# B&R Automation Studio project CControl_Gschneitner (part 15)

#### Main.st - Init, cyclic, exit code
```iecst
PROGRAM _INIT

	hmiStatus.NameSteuerung	:= 6; //= LaTronic CControl 2.07

END_PROGRAM

PROGRAM _CYCLIC

	//Bei Konfiguration 4.07 -> Text auf Login-Seite anpassen, Option Entfeuchter ausschalten

	hmiParameter.Ausstattung.Entfeuchter := FALSE;
	hmiParameter.Ausstattung.Bypassklappe := FALSE;
	hmiParameter.Ausstattung.Box3 := FALSE;
	hmiParameter.Ausstattung.Box4 := FALSE;
	hmiParameter.Ausstattung.Box5 := FALSE;
	hmiParameter.Ausstattung.Box6 := FALSE;

	IF hmiParameter.Ausstattung.Abluftklappe THEN
		hmiParameter.Ausstattung.Abluftventilator := FALSE;
	ELSIF hmiParameter.Ausstattung.Abluftventilator THEN
		hmiParameter.Ausstattung.Abluftklappe := FALSE;
	END_IF

	//Zeitticks generieren
	fbLascoZdxx_0(IN 	:= Echtzeit.Sekunde);
	sekTick				:= fbLascoZdxx_0.Q;

	//=========================================================================================================================================================
	//IO-Zuweisung LaTronic CControl 4.07
	//=========================================================================================================================================================

	//Kein Testbetrieb
	IF (gAktModus <> IOTEST) THEN

		//MODUL 01 - BR7300 Busempfänger **********************************************************************************************************************
		brModul01;

		//MODUL 02 - CM8281 ***********************************************************************************************************************************
		//*****************************************************************************************************************************************************
		diVentilator1InBetrieb	:= cmModul02.di01;
		di24VDCinternIstOk		:= cmModul02.di02;
		//Reserve				:= cmModul02.di03;
		//Reserve				:= cmModul02.di04;

		cmModul02.do01			:= doVentilator1Ein;
		cmModul02.do02			:= doTrocknungInBetrieb;

		//Eingangssignale filtern
		IF sekTick THEN
			LCRMovAvgFlt_0(enable := TRUE, x := cmModul02.ai01, base := Betriebsparameter.Sensoren.FilterzeitFrischluft);
		END_IF

		//Frischluft Temperatur
		LCRLimScal_0(x := LCRMovAvgFlt_0.y, x1 := 0, y1 := Betriebsparameter.Sensoren.FrischlTempMessberMin,
		x2 := 32767, y2 := Betriebsparameter.Sensoren.FrischlTempMessberMax);
		aiFrischluftTemperatur		:= LCRLimScal_0.y + Betriebsparameter.Sensoren.OffsetFrischluftTemp;

		//Drehzahlvorgabe FU Ventilator 1
		LCRLimScal_0(x := aoDrehzahlvorgVentilator1, x1 := Betriebsparameter.Ventilator1.DrehzahlMin, y1 := 0,
		x2 := Betriebsparameter.Ventilator1.DrehzahlMax, y2 := 32767);
		cmModul02.ao01				:= REAL_TO_INT(LCRLimScal_0.y);

		//MODUL 03 - CM8281 ***********************************************************************************************************************************
		//*****************************************************************************************************************************************************
		diBox1Offen				:= cmModul03.di01;
		diBox1Geschl			:= cmModul03.di02;
		diBox2Offen				:= cmModul03.di03;
		diBox2Geschl			:= cmModul03.di04;

		cmModul03.do01			:= doFreigabeBox1;
		cmModul03.do02			:= doFreigabeBox2;

		//Eingangssignale filtern
		IF sekTick THEN
			LCRMovAvgFlt_1(enable := TRUE, x := cmModul03.ai01, base := Betriebsparameter.Sensoren.FilterzeitFrischluft);
		END_IF

		//Frischluft rel. Feuchte
		LCRLimScal_0(x := LCRMovAvgFlt_1.y, x1 := 0, y1 := Betriebsparameter.Sensoren.FrischlFeuchteMessberMin,
		x2 := 32767, y2 := Betriebsparameter.Sensoren.FrischlFeuchteMessberMax);
		aiFrischluftFeuchte		:= LCRLimScal_0.y + Betriebsparameter.Sensoren.OffsetFrischluftFeuchte;

		//Temperaturvorgabe Warmluftofen
		LCRLimScal_0(x := aoTemperaturvorgWarmluftofen, x1 := 0, y1 := 0,
		x2 := 100, y2 := 32767);
		cmModul03.ao01				:= REAL_TO_INT(LCRLimScal_0.y);

		//MODUL 04 - CM8281 ***********************************************************************************************************************************
		//*****************************************************************************************************************************************************
		diVentilator2InBetrieb			:= cmModul04.di01;
		diDrehzahlbegrVentilator1		:= cmModul04.di02;
		diDrehzahlbegrVentilator2		:= cmModul04.di03;
		//Reserve						:= cmModul04.di04;

		cmModul04.do01					:= doTrocknungStoerung;
		cmModul04.do02					:= doVentilator2Ein;

		//Eingangssignale filtern
		IF sekTick THEN
			LCRMovAvgFlt_2(enable := TRUE, x := cmModul04.ai01, base := Betriebsparameter.Sensoren.FilterzeitTrockenluft);
		END_IF

		//Trockenluft Temperatur
		LCRLimScal_0(x := LCRMovAvgFlt_2.y, x1 := 0, y1 := Betriebsparameter.Sensoren.TrockenlTempMessberMin,
		x2 := 32767, y2 := Betriebsparameter.Sensoren.TrockenlTempMessberMax);
		aiTrockenluftTemperatur		:= LCRLimScal_0.y + Betriebsparameter.Sensoren.OffsetTrockenluftTemp;

		//Drehzahlvorgabe FU Ventilator 2
		LCRLimScal_0(x := aoDrehzahlvorgVentilator2, x1 := Betriebsparameter.Ventilator2.DrehzahlMin, y1 := 0,
		x2 := Betriebsparameter.Ventilator2.DrehzahlMax, y2 := 32767);
		cmModul04.ao01				:= REAL_TO_INT(LCRLimScal_0.y);

		//MODUL 05 - CM8281 ***********************************************************************************************************************************
		//*****************************************************************************************************************************************************
		diWarmluftofenInBetrieb		:= cmModul05.di01;
		diScheitholzofenInBetrieb	:= cmModul05.di02;
		//Reserve					:= cmModul05.di03;
		//Reserve					:= cmModul05.di04;

		cmModul05.do01				:= doWarmluftofenEin;
		cmModul05.do02				:= doHeizregisterEin;

		//Eingangssignale filtern
		IF sekTick THEN
			LCRMovAvgFlt_3(enable := TRUE, x := cmModul05.ai01, base := Betriebsparameter.Sensoren.FilterzeitTrockenluft);
		END_IF

		//Trockenluft rel. Feuchte
		LCRLimScal_0(x := LCRMovAvgFlt_3.y, x1 := 0, y1 := Betriebsparameter.Sensoren.TrockenlFeuchteMessberMin,
		x2 := 32767, y2 := Betriebsparameter.Sensoren.TrockenlFeuchteMessberMax);
		aiTrockenluftFeuchte		:= LCRLimScal_0.y + Betriebsparameter.Sensoren.OffsetTrockenluftFeuchte;

		//Leistungsvorgabe Heizregister
		LCRLimScal_0(x := aoLeistungsvorgHeizregister, x1 := 0.0, y1 := 0, x2 := 100.0, y2 := 32767);
		cmModul05.ao01				:= REAL_TO_INT(LCRLimScal_0.y);

		//MODUL 06 - CM8281 ***********************************************************************************************************************************
		//*****************************************************************************************************************************************************
		diBox3Offen				:= cmModul06.di01;
		diBox3Geschl			:= cmModul06.di02;
		diBox4Offen				:= cmModul06.di03;
		diBox4Geschl			:= cmModul06.di04;

		cmModul06.do01			:= doFreigabeBox3;
		cmModul06.do02			:= doFreigabeBox4;

		//Eingangssignale filtern
		IF sekTick THEN
			LCRMovAvgFlt_4(enable := TRUE, x := cmModul06.ai01, base := Betriebsparameter.Sensoren.FilterzeitAbluft);
		END_IF

		//Abluft Temperatur
		LCRLimScal_0(x := LCRMovAvgFlt_4.y, x1 := 0, y1 := Betriebsparameter.Sensoren.AbluftTempMessberMin,
		x2 := 32767, y2 := Betriebsparameter.Sensoren.AbluftTempMessberMax);
		aiAbluftTemperatur		:= LCRLimScal_0.y + Betriebsparameter.Sensoren.OffsetAbluftTemp;

		//Analogausgang
		cmModul06.ao01				:= 0;	//Reserve

		//MODUL 07 - CM8281 ***********************************************************************************************************************************
		//*****************************************************************************************************************************************************
		diBox5Offen				:= cmModul07.di01;
		diBox5Geschl			:= cmModul07.di02;
		diBox6Offen				:= cmModul07.di03;
		diBox6Geschl			:= cmModul07.di04;

		cmModul07.do01			:= doFreigabeBox5;
		cmModul07.do02			:= doFreigabeBox6;

		//Eingangssignale filtern
		IF sekTick THEN
			LCRMovAvgFlt_5(enable := TRUE, x := cmModul07.ai01, base := Betriebsparameter.Sensoren.FilterzeitAbluft);
		END_IF

		//Abluft rel. Feuchte
		LCRLimScal_0(x := LCRMovAvgFlt_5.y, x1 := 0, y1 := Betriebsparameter.Sensoren.AbluftFeuchteMessberMin,
		x2 := 32767, y2 := Betriebsparameter.Sensoren.AbluftFeuchteMessberMax);
		aiAbluftFeuchte		:= LCRLimScal_0.y + Betriebsparameter.Sensoren.OffsetAbluftFeuchte;

		//Analogausgang
		cmModul07.ao01				:= 0;	//Reserve

		//MODUL 08 - CM8281 ***********************************************************************************************************************************
		//*****************************************************************************************************************************************************
		diAbluftventInBetrieb	:= cmModul08.di01;
		//Reserve				:= cmModul08.di02;
		//Reserve				:= cmModul08.di03;
		//Reserve				:= cmModul08.di04;

		cmModul08.do01			:= doBrandschutzklappeAuf;
		cmModul08.do02			:= doAbluftventilatorEin;

		//Eingangssignale filtern
		IF sekTick THEN
			LCRMovAvgFlt_6(enable := TRUE, x := cmModul08.ai01, base := Betriebsparameter.Sensoren.FilterzeitDachluft);
		END_IF

		//Dachluft Temperatur
		LCRLimScal_0(x := LCRMovAvgFlt_6.y, x1 := 0, y1 := Betriebsparameter.Sensoren.DachTempMessberMin,
		x2 := 32767, y2 := Betriebsparameter.Sensoren.DachTempMessberMax);
		aiDachluftTemperatur		:= LCRLimScal_0.y + Betriebsparameter.Sensoren.OffsetDachTemp;

		//Drehzahlvorgabe Abluftventilator
		LCRLimScal_0(x := aoDrehzahlvorgAbluftventilator, x1 := Betriebsparameter.Abluftventilator.DrehzahlMin, y1 := 0,
		x2 := Betriebsparameter.Abluftventilator.DrehzahlMax, y2 := 32767);
		cmModul08.ao01				:= REAL_TO_INT(LCRLimScal_0.y);

		//MODUL 09 - CM8281 ***********************************************************************************************************************************
		//*****************************************************************************************************************************************************
		diAbluftklappeOffen		:= cmModul09.di01;
		diAbluftklappeGeschl	:= cmModul09.di02;
		//Reserve				:= cmModul09.di03;
		//Reserve				:= cmModul09.di04;

		cmModul09.do01			:= doAbluftklappeFreigabe;
		cmModul09.do02			:= FALSE;	//Reserve

		//Eingangssignale filtern
		IF sekTick THEN
			LCRMovAvgFlt_7(enable := TRUE, x := cmModul09.ai01, base := Betriebsparameter.Sensoren.FilterzeitDachluft);
		END_IF

		//Dachluft rel. Feuchte
		LCRLimScal_0(x := LCRMovAvgFlt_7.y, x1 := 0, y1 := Betriebsparameter.Sensoren.DachFeuchteMessberMin,
		x2 := 32767, y2 := Betriebsparameter.Sensoren.DachFeuchteMessberMax);
		aiDachluftFeuchte		:= LCRLimScal_0.y + Betriebsparameter.Sensoren.OffsetDachFeuchte;

		//Analogausgang
		cmModul09.ao01				:= 0;	//Reserve

		//MODUL 10 - CM8281 ***********************************************************************************************************************************
		//*****************************************************************************************************************************************************
		diUmschaltklappe1Offen		:= cmModul10.di01;
		diUmschaltklappe1Geschl		:= cmModul10.di02;
		diUmschaltklappe2Offen		:= cmModul10.di03;
		diUmschaltklappe2Geschl		:= cmModul10.di04;

		cmModul10.do01				:= doUmluftklappe1Freigabe;
		cmModul10.do02				:= doUmluftklappe2Freigabe;

		//Eingangssignale filtern
		IF sekTick THEN
			LCRMovAvgFlt_8(enable := TRUE, x := cmModul10.ai01, base := Betriebsparameter.Sensoren.FilterzeitLuftgeschwindigkeit);
		END_IF

		//Luftgeschwindigkeit
		LCRLimScal_0(x := LCRMovAvgFlt_8.y, x1 := 0, y1 := Betriebsparameter.Sensoren.LuftgeschwMessberMin,
		x2 := 32767, y2 := Betriebsparameter.Sensoren.LuftgeschwMessberMax);
		aiLuftgeschwindigkeit		:= LCRLimScal_0.y + Betriebsparameter.Sensoren.OffsetLuftgeschw;

		//Analogausgang
		cmModul10.ao01				:= 0;	//Reserve

		//MODUL 11 - CM8281 ***********************************************************************************************************************************
		//*****************************************************************************************************************************************************
		diNotstromaggregatInBetrieb		:= cmModul11.di01;
		//Reserve						:= cmModul11.di02;
		//Reserve						:= cmModul11.di03;
		//Reserve						:= cmModul11.di04;

		cmModul11.do01					:= doNotstromaggregatEin;
		cmModul11.do02					:= FALSE;	//Reserve

		//Eingangssignale filtern
		IF sekTick THEN
			LCRMovAvgFlt_9(enable := TRUE, x := cmModul11.ai01, base := Betriebsparameter.Sensoren.FilterzeitKanaldruck);
		END_IF

		//Differenzdruck
		LCRLimScal_0(x := LCRMovAvgFlt_9.y, x1 := 0, y1 := Betriebsparameter.Sensoren.KanaldruckMessberMin,
		x2 := 32767, y2 := Betriebsparameter.Sensoren.KanaldruckMessberMax);
		aiDifferenzdruck		:= LCRLimScal_0.y + Betriebsparameter.Sensoren.OffsetKanaldruck;

		//Analogausgang
		cmModul11.ao01				:= 0;	//Reserve

		//Modulstatus - Auswertung **********************************************************************************************************************************
		//***********************************************************************************************************************************************************

		//Modul 02 Frischluft Temperatur ****************************************************************************
		IF (cmModul02.StatusInput01.1 = FALSE AND cmModul02.StatusInput01.0 = TRUE) THEN
			diStatusFrischluftTempMin	:= TRUE;
		ELSE
			diStatusFrischluftTempMin	:= FALSE;
		END_IF
		IF (cmModul02.StatusInput01.1 = TRUE AND cmModul02.StatusInput01.0 = FALSE ) THEN
			diStatusFrischluftTempMax	 := TRUE;
		ELSE
			diStatusFrischluftTempMax	 := FALSE;
		END_IF

		//Modul 03 Frischluft rel. Feuchte ****************************************************************************
		IF (cmModul03.StatusInput01.1 = FALSE AND cmModul03.StatusInput01.0 = TRUE) THEN
			diStatusFrischluftFeuchteMin	:= TRUE;
		ELSE
			diStatusFrischluftFeuchteMin	:= FALSE;
		END_IF
		IF (cmModul03.StatusInput01.1 = TRUE AND cmModul03.StatusInput01.0 = FALSE ) THEN
			diStatusFrischluftFeuchteMax	 := TRUE;
		ELSE
			diStatusFrischluftFeuchteMax	 := FALSE;
		END_IF

		//Modul 04 Trockenluft Temperatur ****************************************************************************
		IF (cmModul04.StatusInput01.1 = FALSE AND cmModul04.StatusInput01.0 = TRUE) THEN
			diStatusTrockenluftTempMin	:= TRUE;
		ELSE
			diStatusTrockenluftTempMin	:= FALSE;
		END_IF
		IF (cmModul04.StatusInput01.1 = TRUE AND cmModul04.StatusInput01.0 = FALSE ) THEN
			diStatusTrockenluftTempMax	 := TRUE;
		ELSE
			diStatusTrockenluftTempMax	 := FALSE;
		END_IF

		//Modul 05 Trockenluft rel. Feuchte ****************************************************************************
		IF (cmModul05.StatusInput01.1 = FALSE AND cmModul05.StatusInput01.0 = TRUE) THEN
			diStatusTrockenluftFeuchteMin	:= TRUE;
		ELSE
			diStatusTrockenluftFeuchteMin	:= FALSE;
		END_IF
		IF (cmModul05.StatusInput01.1 = TRUE AND cmModul05.StatusInput01.0 = FALSE ) THEN
			diStatusTrockenluftFeuchteMax	 := TRUE;
		ELSE
			diStatusTrockenluftFeuchteMax	 := FALSE;
		END_IF

		//Modul 06 Abluft Temperatur ****************************************************************************
		IF (cmModul06.StatusInput01.1 = FALSE AND cmModul06.StatusInput01.0 = TRUE) THEN
			diStatusAbluftTempMin	:= TRUE;
		ELSE
			diStatusAbluftTempMin	:= FALSE;
		END_IF
		IF (cmModul06.StatusInput01.1 = TRUE AND cmModul06.StatusInput01.0 = FALSE ) THEN
			diStatusAbluftTempMax	 := TRUE;
		ELSE
			diStatusAbluftTempMax	 := FALSE;
		END_IF

		//Modul 07 Abluft rel. Feuchte ****************************************************************************
		IF (cmModul07.StatusInput01.1 = FALSE AND cmModul07.StatusInput01.0 = TRUE) THEN
			diStatusAbluftFeuchteMin	:= TRUE;
		ELSE
			diStatusAbluftFeuchteMin	:= FALSE;
		END_IF
		IF (cmModul07.StatusInput01.1 = TRUE AND cmModul07.StatusInput01.0 = FALSE ) THEN
			diStatusAbluftFeuchteMax	 := TRUE;
		ELSE
			diStatusAbluftFeuchteMax	 := FALSE;
		END_IF

		//Modul 08 Dachluft Temperatur ****************************************************************************
		IF (cmModul08.StatusInput01.1 = FALSE AND cmModul08.StatusInput01.0 = TRUE) THEN
			diStatusDachluftTempMin	:= TRUE;
		ELSE
			diStatusDachluftTempMin	:= FALSE;
		END_IF
		IF (cmModul08.StatusInput01.1 = TRUE AND cmModul08.StatusInput01.0 = FALSE ) THEN
			diStatusDachluftTempMax	 := TRUE;
		ELSE
			diStatusDachluftTempMax	 := FALSE;
		END_IF

		//Modul 09 Dachluft rel. Feuchte ****************************************************************************
		IF (cmModul09.StatusInput01.1 = FALSE AND cmModul09.StatusInput01.0 = TRUE) THEN
			diStatusDachluftFeuchteMin	:= TRUE;
		ELSE
			diStatusDachluftFeuchteMin	:= FALSE;
		END_IF
		IF (cmModul09.StatusInput01.1 = TRUE AND cmModul09.StatusInput01.0 = FALSE ) THEN
			diStatusDachluftFeuchteMax	 := TRUE;
		ELSE
			diStatusDachluftFeuchteMax	 := FALSE;
		END_IF

		//Modul 10 Luftgeschwindigkeit ****************************************************************************
		IF (cmModul10.StatusInput01.1 = FALSE AND cmModul10.StatusInput01.0 = TRUE) THEN
			diStatusLuftgeschwMin	:= TRUE;
		ELSE
			diStatusLuftgeschwMin	:= FALSE;
		END_IF
		IF (cmModul10.StatusInput01.1 = TRUE AND cmModul10.StatusInput01.0 = FALSE ) THEN
			diStatusLuftgeschwMax	:= TRUE;
		ELSE
			diStatusLuftgeschwMax	 := FALSE;
		END_IF
		IF ((cmModul10.StatusInput01.1 = TRUE AND cmModul10.StatusInput01.0 = TRUE) OR cmModul10.ai01 >= 32767) THEN
			diStatusLuftgeschwDrahtbruch := TRUE;
		ELSE
			diStatusLuftgeschwDrahtbruch := FALSE;
		END_IF

		//Modul 11 Differenzdruck ****************************************************************************
		IF (cmModul11.StatusInput01.1 = FALSE AND cmModul11.StatusInput01.0 = TRUE) THEN
			diStatusDifferenzdruckMin	:= TRUE;
		ELSE
			diStatusDifferenzdruckMin	:= FALSE;
		END_IF
		IF (cmModul11.StatusInput01.1 = TRUE AND cmModul11.StatusInput01.0 = FALSE ) THEN
			diStatusDifferenzdruckMax	 := TRUE;
		ELSE
			diStatusDifferenzdruckMax	 := FALSE;
		END_IF

		//Ausgänge Testbetrieb rücksetzen, wenn IO-Test nicht aktiv
		hmiIoTest.DigitalOut.doAbluftklappeFreigabe		:= FALSE;
		hmiIoTest.DigitalOut.doAbluftventilatorEin		:= FALSE;
		hmiIoTest.DigitalOut.doBrandschutzklappeAuf		:= FALSE;
		hmiIoTest.DigitalOut.doBypassklappeOeffnen		:= FALSE;
		hmiIoTest.DigitalOut.doFreigabeBox1				:= FALSE;
		hmiIoTest.DigitalOut.doFreigabeBox2				:= FALSE;
		hmiIoTest.DigitalOut.doFreigabeBox3				:= FALSE;
		hmiIoTest.DigitalOut.doFreigabeBox4				:= FALSE;
		hmiIoTest.DigitalOut.doFreigabeBox5				:= FALSE;
		hmiIoTest.DigitalOut.doFreigabeBox6				:= FALSE;
		hmiIoTest.DigitalOut.doHeizregisterEin			:= FALSE;
		hmiIoTest.DigitalOut.doKompressorEinModul1		:= FALSE;
		hmiIoTest.DigitalOut.doKompressorEinModul2		:= FALSE;
		hmiIoTest.DigitalOut.doMagnetventilEinModul1	:= FALSE;
		hmiIoTest.DigitalOut.doMagnetventilEinModul2	:= FALSE;
		hmiIoTest.DigitalOut.doNotstromaggregatEin		:= FALSE;
		hmiIoTest.DigitalOut.doOelsumpfheizungEinModul1	:= FALSE;
		hmiIoTest.DigitalOut.doOelsumpfheizungEinModul2	:= FALSE;
		hmiIoTest.DigitalOut.doTrocknungInBetrieb		:= FALSE;
		hmiIoTest.DigitalOut.doTrocknungStoerung		:= FALSE;
		hmiIoTest.DigitalOut.doUmluftklappe1Freigabe	:= FALSE;
		hmiIoTest.DigitalOut.doUmluftklappe2Freigabe	:= FALSE;
		hmiIoTest.DigitalOut.doVentilator1Ein			:= FALSE;
		hmiIoTest.DigitalOut.doVentilator2Ein			:= FALSE;
		hmiIoTest.DigitalOut.doWarmluftofenEin			:= FALSE;

		hmiIoTest.AnalogOut.aoDrehzahlvorgAbluftventilator	:= 0.0;
		hmiIoTest.AnalogOut.aoDrehzahlvorgKompressorModul1	:= 0.0;
		hmiIoTest.AnalogOut.aoDrehzahlvorgKompressorModul2	:= 0.0;
		hmiIoTest.AnalogOut.aoDrehzahlvorgVentilator1		:= 0.0;
		hmiIoTest.AnalogOut.aoDrehzahlvorgVentilator2		:= 0.0;
		hmiIoTest.AnalogOut.aoLeistungsvorgHeizregister		:= 0.0;
		hmiIoTest.AnalogOut.aoTemperaturvorgWarmluftofen	:= 0.0;

	//==============================================================================================================================================================================================================
	//Testbetrieb
	//==============================================================================================================================================================================================================
	ELSE

		//MODUL 01 - BR7300 Busempfänger **********************************************************************************************************************

		//MODUL 02 - CM8281 ***********************************************************************************************************************************
		//*****************************************************************************************************************************************************
		hmiIoTest.DigitalIn.diVentilator1InBetrieb	:= cmModul02.di01;
		hmiIoTest.DigitalIn.di24VDCinternIstOk		:= cmModul02.di02;
		//Reserve									:= cmModul02.di03;
		//Reserve									:= cmModul02.di04;

		cmModul02.do01			:= hmiIoTest.DigitalOut.doVentilator1Ein;
		cmModul02.do02			:= hmiIoTest.DigitalOut.doTrocknungInBetrieb;

		//Eingangssignale filtern
		IF sekTick THEN
			LCRMovAvgFlt_0(enable := TRUE, x := cmModul02.ai01, base := Betriebsparameter.Sensoren.FilterzeitFrischluft);
		END_IF

		//Frischluft Temperatur
		LCRLimScal_0(x := LCRMovAvgFlt_0.y, x1 := 0, y1 := Betriebsparameter.Sensoren.FrischlTempMessberMin,
		x2 := 32767, y2 := Betriebsparameter.Sensoren.FrischlTempMessberMax);
		hmiIoTest.AnalogIn.aiFrischluftTemperatur		:= LCRLimScal_0.y + Betriebsparameter.Sensoren.OffsetFrischluftTemp;

		//Drehzahlvorgabe FU Ventilator 1
		LCRLimScal_0(x := hmiIoTest.AnalogOut.aoDrehzahlvorgVentilator1, x1 := Betriebsparameter.Ventilator1.DrehzahlMin, y1 := 0,
		x2 := Betriebsparameter.Ventilator1.DrehzahlMax, y2 := 32767);
		cmModul02.ao01				:= REAL_TO_INT(LCRLimScal_0.y);

		//MODUL 03 - CM8281 ***********************************************************************************************************************************
		//*****************************************************************************************************************************************************
		hmiIoTest.DigitalIn.diBox1Offen				:= cmModul03.di01;
		hmiIoTest.DigitalIn.diBox1Geschl			:= cmModul03.di02;
		hmiIoTest.DigitalIn.diBox2Offen				:= cmModul03.di03;
		hmiIoTest.DigitalIn.diBox2Geschl			:= cmModul03.di04;

		cmModul03.do01			:= hmiIoTest.DigitalOut.doFreigabeBox1;
		cmModul03.do02			:= hmiIoTest.DigitalOut.doFreigabeBox2;

		//Eingangssignale filtern
		IF sekTick THEN
			LCRMovAvgFlt_1(enable := TRUE, x := cmModul03.ai01, base := Betriebsparameter.Sensoren.FilterzeitFrischluft);
		END_IF

		//Frischluft rel. Feuchte
		LCRLimScal_0(x := LCRMovAvgFlt_1.y, x1 := 0, y1 := Betriebsparameter.Sensoren.FrischlFeuchteMessberMin,
		x2 := 32767, y2 := Betriebsparameter.Sensoren.FrischlFeuchteMessberMax);
		hmiIoTest.AnalogIn.aiFrischluftFeuchte		:= LCRLimScal_0.y + Betriebsparameter.Sensoren.OffsetFrischluftFeuchte;

		//Temperaturvorgabe Warmluftofen
		LCRLimScal_0(x := hmiIoTest.AnalogOut.aoTemperaturvorgWarmluftofen, x1 := 0, y1 := 0,
		x2 := 100, y2 := 32767);
		cmModul03.ao01				:= REAL_TO_INT(LCRLimScal_0.y);

		//MODUL 04 - CM8281 ***********************************************************************************************************************************
		//*****************************************************************************************************************************************************
		hmiIoTest.DigitalIn.diVentilator2InBetrieb			:= cmModul04.di01;
		hmiIoTest.DigitalIn.diDrehzahlbegrVentilator1		:= cmModul04.di02;
		hmiIoTest.DigitalIn.diDrehzahlbegrVentilator2		:= cmModul04.di03;
		//Reserve											:= cmModul04.di04;

		cmModul04.do01					:= hmiIoTest.DigitalOut.doTrocknungStoerung;
		cmModul04.do02					:= hmiIoTest.DigitalOut.doVentilator2Ein;

		//Eingangssignale filtern
		IF sekTick THEN
			LCRMovAvgFlt_2(enable := TRUE, x := cmModul04.ai01, base := Betriebsparameter.Sensoren.FilterzeitTrockenluft);
		END_IF

		//Trockenluft Temperatur
		LCRLimScal_0(x := LCRMovAvgFlt_2.y, x1 := 0, y1 := Betriebsparameter.Sensoren.TrockenlTempMessberMin,
		x2 := 32767, y2 := Betriebsparameter.Sensoren.TrockenlTempMessberMax);
		hmiIoTest.AnalogIn.aiTrockenluftTemperatur		:= LCRLimScal_0.y + Betriebsparameter.Sensoren.OffsetTrockenluftTemp;

		//Drehzahlvorgabe FU Ventilator 2
		LCRLimScal_0(x := hmiIoTest.AnalogOut.aoDrehzahlvorgVentilator2, x1 := Betriebsparameter.Ventilator2.DrehzahlMin, y1 := 0,
		x2 := Betriebsparameter.Ventilator2.DrehzahlMax, y2 := 32767);
		cmModul04.ao01				:= REAL_TO_INT(LCRLimScal_0.y);

		//MODUL 05 - CM8281 ***********************************************************************************************************************************
		//*****************************************************************************************************************************************************
		hmiIoTest.DigitalIn.diWarmluftofenInBetrieb		:= cmModul05.di01;
		hmiIoTest.DigitalIn.diScheitholzofenInBetrieb	:= cmModul05.di02;
		//Reserve										:= cmModul05.di03;
		//Reserve										:= cmModul05.di04;

		cmModul05.do01				:= hmiIoTest.DigitalOut.doWarmluftofenEin;
		cmModul05.do02				:= hmiIoTest.DigitalOut.doHeizregisterEin;

		//Eingangssignale filtern
		IF sekTick THEN
			LCRMovAvgFlt_3(enable := TRUE, x := cmModul05.ai01, base := Betriebsparameter.Sensoren.FilterzeitTrockenluft);
		END_IF

		//Trockenluft rel. Feuchte
		LCRLimScal_0(x := LCRMovAvgFlt_3.y, x1 := 0, y1 := Betriebsparameter.Sensoren.TrockenlFeuchteMessberMin,
		x2 := 32767, y2 := Betriebsparameter.Sensoren.TrockenlFeuchteMessberMax);
		hmiIoTest.AnalogIn.aiTrockenluftFeuchte		:= LCRLimScal_0.y + Betriebsparameter.Sensoren.OffsetTrockenluftFeuchte;

		//Leistungsvorgabe Heizregister
		LCRLimScal_0(x := hmiIoTest.AnalogOut.aoLeistungsvorgHeizregister, x1 := 0.0, y1 := 0, x2 := 100.0, y2 := 32767);
		cmModul05.ao01				:= REAL_TO_INT(LCRLimScal_0.y);

		//MODUL 06 - CM8281 ***********************************************************************************************************************************
		//*****************************************************************************************************************************************************
		hmiIoTest.DigitalIn.diBox3Offen				:= cmModul06.di01;
		hmiIoTest.DigitalIn.diBox3Geschl			:= cmModul06.di02;
		hmiIoTest.DigitalIn.diBox4Offen				:= cmModul06.di03;
		hmiIoTest.DigitalIn.diBox4Geschl			:= cmModul06.di04;

		cmModul06.do01			:= hmiIoTest.DigitalOut.doFreigabeBox3;
		cmModul06.do02			:= hmiIoTest.DigitalOut.doFreigabeBox4;

		//Eingangssignale filtern
		IF sekTick THEN
			LCRMovAvgFlt_4(enable := TRUE, x := cmModul06.ai01, base := Betriebsparameter.Sensoren.FilterzeitAbluft);
		END_IF

		//Abluft Temperatur
		LCRLimScal_0(x := LCRMovAvgFlt_4.y, x1 := 0, y1 := Betriebsparameter.Sensoren.AbluftTempMessberMin,
		x2 := 32767, y2 := Betriebsparameter.Sensoren.AbluftTempMessberMax);
		hmiIoTest.AnalogIn.aiAbluftTemperatur		:= LCRLimScal_0.y + Betriebsparameter.Sensoren.OffsetAbluftTemp;

		//Analogausgang
		cmModul06.ao01				:= 0;	//Reserve

		//MODUL 07 - CM8281 ***********************************************************************************************************************************
		//*****************************************************************************************************************************************************
		hmiIoTest.DigitalIn.diBox5Offen				:= cmModul07.di01;
		hmiIoTest.DigitalIn.diBox5Geschl			:= cmModul07.di02;
		hmiIoTest.DigitalIn.diBox6Offen				:= cmModul07.di03;
		hmiIoTest.DigitalIn.diBox6Geschl			:= cmModul07.di04;

		cmModul07.do01			:= hmiIoTest.DigitalOut.doFreigabeBox5;
		cmModul07.do02			:= hmiIoTest.DigitalOut.doFreigabeBox6;

		//Eingangssignale filtern
		IF sekTick THEN
			LCRMovAvgFlt_5(enable := TRUE, x := cmModul07.ai01, base := Betriebsparameter.Sensoren.FilterzeitAbluft);
		END_IF

		//Abluft rel. Feuchte
		LCRLimScal_0(x := LCRMovAvgFlt_5.y, x1 := 0, y1 := Betriebsparameter.Sensoren.AbluftFeuchteMessberMin,
		x2 := 32767, y2 := Betriebsparameter.Sensoren.AbluftFeuchteMessberMax);
		hmiIoTest.AnalogIn.aiAbluftFeuchte		:= LCRLimScal_0.y + Betriebsparameter.Sensoren.OffsetAbluftFeuchte;

		//Analogausgang
		cmModul07.ao01				:= 0;	//Reserve

		//MODUL 08 - CM8281 ***********************************************************************************************************************************
		//*****************************************************************************************************************************************************
		hmiIoTest.DigitalIn.diAbluftventInBetrieb	:= cmModul08.di01;
		//Reserve									:= cmModul08.di02;
		//Reserve									:= cmModul08.di03;
		//Reserve									:= cmModul08.di04;

		cmModul08.do01			:= hmiIoTest.DigitalOut.doBrandschutzklappeAuf;
		cmModul08.do02			:= hmiIoTest.DigitalOut.doAbluftventilatorEin;

		//Eingangssignale filtern
		IF sekTick THEN
			LCRMovAvgFlt_6(enable := TRUE, x := cmModul08.ai01, base := Betriebsparameter.Sensoren.FilterzeitDachluft);
		END_IF

		//Dachluft Temperatur
		LCRLimScal_0(x := LCRMovAvgFlt_6.y, x1 := 0, y1 := Betriebsparameter.Sensoren.DachTempMessberMin,
		x2 := 32767, y2 := Betriebsparameter.Sensoren.DachTempMessberMax);
		hmiIoTest.AnalogIn.aiDachluftTemperatur		:= LCRLimScal_0.y + Betriebsparameter.Sensoren.OffsetDachTemp;

		//Drehzahlvorgabe Abluftventilator
		LCRLimScal_0(x := hmiIoTest.AnalogOut.aoDrehzahlvorgAbluftventilator, x1 := Betriebsparameter.Abluftventilator.DrehzahlMin, y1 := 0,
		x2 := Betriebsparameter.Abluftventilator.DrehzahlMax, y2 := 32767);
		cmModul08.ao01				:= REAL_TO_INT(LCRLimScal_0.y);

		//MODUL 09 - CM8281 ***********************************************************************************************************************************
		//*****************************************************************************************************************************************************
		hmiIoTest.DigitalIn.diAbluftklappeOffen		:= cmModul09.di01;
		hmiIoTest.DigitalIn.diAbluftklappeGeschl	:= cmModul09.di02;
		//Reserve									:= cmModul09.di03;
		//Reserve									:= cmModul09.di04;

		cmModul09.do01			:= hmiIoTest.DigitalOut.doAbluftklappeFreigabe;
		cmModul09.do02			:= FALSE;	//Reserve

		//Eingangssignale filtern
		IF sekTick THEN
			LCRMovAvgFlt_7(enable := TRUE, x := cmModul09.ai01, base := Betriebsparameter.Sensoren.FilterzeitDachluft);
		END_IF

		//Dachluft rel. Feuchte
		LCRLimScal_0(x := LCRMovAvgFlt_7.y, x1 := 0, y1 := Betriebsparameter.Sensoren.DachFeuchteMessberMin,
		x2 := 32767, y2 := Betriebsparameter.Sensoren.DachFeuchteMessberMax);
		hmiIoTest.AnalogIn.aiDachluftFeuchte		:= LCRLimScal_0.y + Betriebsparameter.Sensoren.OffsetDachFeuchte;

		//Analogausgang
		cmModul09.ao01				:= 0;	//Reserve

		//MODUL 10 - CM8281 ***********************************************************************************************************************************
		//*****************************************************************************************************************************************************
		hmiIoTest.DigitalIn.diUmschaltklappe1Offen		:= cmModul10.di01;
		hmiIoTest.DigitalIn.diUmschaltklappe1Geschl		:= cmModul10.di02;
		hmiIoTest.DigitalIn.diUmschaltklappe2Offen		:= cmModul10.di03;
		hmiIoTest.DigitalIn.diUmschaltklappe2Geschl		:= cmModul10.di04;

		cmModul10.do01				:= hmiIoTest.DigitalOut.doUmluftklappe1Freigabe;
		cmModul10.do02				:= hmiIoTest.DigitalOut.doUmluftklappe2Freigabe;

		//Eingangssignale filtern
		IF sekTick THEN
			LCRMovAvgFlt_8(enable := TRUE, x := cmModul10.ai01, base := Betriebsparameter.Sensoren.FilterzeitLuftgeschwindigkeit);
		END_IF

		//Luftgeschwindigkeit
		LCRLimScal_0(x := LCRMovAvgFlt_8.y, x1 := 0, y1 := Betriebsparameter.Sensoren.LuftgeschwMessberMin,
		x2 := 32767, y2 := Betriebsparameter.Sensoren.LuftgeschwMessberMax);
		hmiIoTest.AnalogIn.aiLuftgeschwindigkeit		:= LCRLimScal_0.y + Betriebsparameter.Sensoren.OffsetLuftgeschw;

		//Analogausgang
		cmModul10.ao01				:= 0;	//Reserve

		//MODUL 11 - CM8281 ***********************************************************************************************************************************
		//*****************************************************************************************************************************************************
		hmiIoTest.DigitalIn.diNotstromaggregatInBetrieb		:= cmModul11.di01;
		//Reserve											:= cmModul11.di02;
		//Reserve											:= cmModul11.di03;
		//Reserve											:= cmModul11.di04;

		cmModul11.do01					:= hmiIoTest.DigitalOut.doNotstromaggregatEin;
		cmModul11.do02					:= FALSE;	//Reserve

		//Eingangssignale filtern
		IF sekTick THEN
			LCRMovAvgFlt_9(enable := TRUE, x := cmModul11.ai01, base := Betriebsparameter.Sensoren.FilterzeitKanaldruck);
		END_IF

		//Differenzdruck
		LCRLimScal_0(x := LCRMovAvgFlt_9.y, x1 := 0, y1 := Betriebsparameter.Sensoren.KanaldruckMessberMin,
		x2 := 32767, y2 := Betriebsparameter.Sensoren.KanaldruckMessberMax);
		hmiIoTest.AnalogIn.aiDifferenzdruck		:= LCRLimScal_0.y + Betriebsparameter.Sensoren.OffsetKanaldruck;

		//Analogausgang
		cmModul11.ao01				:= 0;	//Reserve

		//Modulstatus - Auswertung **********************************************************************************************************************************
		//***********************************************************************************************************************************************************

		//Modul 02 Frischluft Temperatur ****************************************************************************
		IF (cmModul02.StatusInput01.1 = FALSE AND cmModul02.StatusInput01.0 = TRUE) THEN
			hmiIoTest.StatusIn.diStatusFrischluftTempMin	:= TRUE;
		ELSE
			diStatusFrischluftTempMin	:= FALSE;
		END_IF
		IF (cmModul02.StatusInput01.1 = TRUE AND cmModul02.StatusInput01.0 = FALSE ) THEN
			hmiIoTest.StatusIn.diStatusFrischluftTempMax	 := TRUE;
		ELSE
			hmiIoTest.StatusIn.diStatusFrischluftTempMax	 := FALSE;
		END_IF

		//Modul 03 Frischluft rel. Feuchte ****************************************************************************
		IF (cmModul03.StatusInput01.1 = FALSE AND cmModul03.StatusInput01.0 = TRUE) THEN
			hmiIoTest.StatusIn.diStatusFrischluftFeuchteMin	:= TRUE;
		ELSE
			hmiIoTest.StatusIn.diStatusFrischluftFeuchteMin	:= FALSE;
		END_IF
		IF (cmModul03.StatusInput01.1 = TRUE AND cmModul03.StatusInput01.0 = FALSE ) THEN
			hmiIoTest.StatusIn.diStatusFrischluftFeuchteMax	 := TRUE;
		ELSE
			hmiIoTest.StatusIn.diStatusFrischluftFeuchteMax	 := FALSE;
		END_IF

		//Modul 04 Trockenluft Temperatur ****************************************************************************
		IF (cmModul04.StatusInput01.1 = FALSE AND cmModul04.StatusInput01.0 = TRUE) THEN
			hmiIoTest.StatusIn.diStatusTrockenluftTempMin	:= TRUE;
		ELSE
			hmiIoTest.StatusIn.diStatusTrockenluftTempMin	:= FALSE;
		END_IF
		IF (cmModul04.StatusInput01.1 = TRUE AND cmModul04.StatusInput01.0 = FALSE ) THEN
			hmiIoTest.StatusIn.diStatusTrockenluftTempMax	 := TRUE;
		ELSE
			hmiIoTest.StatusIn.diStatusTrockenluftTempMax	 := FALSE;
		END_IF

		//Modul 05 Trockenluft rel. Feuchte ****************************************************************************
		IF (cmModul05.StatusInput01.1 = FALSE AND cmModul05.StatusInput01.0 = TRUE) THEN
			hmiIoTest.StatusIn.diStatusTrockenluftFeuchteMin	:= TRUE;
		ELSE
			hmiIoTest.StatusIn.diStatusTrockenluftFeuchteMin	:= FALSE;
		END_IF
		IF (cmModul05.StatusInput01.1 = TRUE AND cmModul05.StatusInput01.0 = FALSE ) THEN
			hmiIoTest.StatusIn.diStatusTrockenluftFeuchteMax	 := TRUE;
		ELSE
			hmiIoTest.StatusIn.diStatusTrockenluftFeuchteMax	 := FALSE;
		END_IF

		//Modul 06 Abluft Temperatur ****************************************************************************
		IF (cmModul06.StatusInput01.1 = FALSE AND cmModul06.StatusInput01.0 = TRUE) THEN
			hmiIoTest.StatusIn.diStatusAbluftTempMin	:= TRUE;
		ELSE
			hmiIoTest.StatusIn.diStatusAbluftTempMin	:= FALSE;
		END_IF
		IF (cmModul06.StatusInput01.1 = TRUE AND cmModul06.StatusInput01.0 = FALSE ) THEN
			hmiIoTest.StatusIn.diStatusAbluftTempMax	 := TRUE;
		ELSE
			hmiIoTest.StatusIn.diStatusAbluftTempMax	 := FALSE;
		END_IF

		//Modul 07 Abluft rel. Feuchte ****************************************************************************
		IF (cmModul07.StatusInput01.1 = FALSE AND cmModul07.StatusInput01.0 = TRUE) THEN
			hmiIoTest.StatusIn.diStatusAbluftFeuchteMin	:= TRUE;
		ELSE
			hmiIoTest.StatusIn.diStatusAbluftFeuchteMin	:= FALSE;
		END_IF
		IF (cmModul07.StatusInput01.1 = TRUE AND cmModul07.StatusInput01.0 = FALSE ) THEN
			hmiIoTest.StatusIn.diStatusAbluftFeuchteMax	 := TRUE;
		ELSE
			hmiIoTest.StatusIn.diStatusAbluftFeuchteMax	 := FALSE;
		END_IF

		//Modul 08 Dachluft Temperatur ****************************************************************************
		IF (cmModul08.StatusInput01.1 = FALSE AND cmModul08.StatusInput01.0 = TRUE) THEN
			hmiIoTest.StatusIn.diStatusDachluftTempMin	:= TRUE;
		ELSE
			hmiIoTest.StatusIn.diStatusDachluftTempMin	:= FALSE;
		END_IF
		IF (cmModul08.StatusInput01.1 = TRUE AND cmModul08.StatusInput01.0 = FALSE ) THEN
			hmiIoTest.StatusIn.diStatusDachluftTempMax	 := TRUE;
		ELSE
			hmiIoTest.StatusIn.diStatusDachluftTempMax	 := FALSE;
		END_IF

		//Modul 09 Dachluft rel. Feuchte ****************************************************************************
		IF (cmModul09.StatusInput01.1 = FALSE AND cmModul09.StatusInput01.0 = TRUE) THEN
			hmiIoTest.StatusIn.diStatusDachluftFeuchteMin	:= TRUE;
		ELSE
			hmiIoTest.StatusIn.diStatusDachluftFeuchteMin	:= FALSE;
		END_IF
		IF (cmModul09.StatusInput01.1 = TRUE AND cmModul09.StatusInput01.0 = FALSE ) THEN
			hmiIoTest.StatusIn.diStatusDachluftFeuchteMax	 := TRUE;
		ELSE
			hmiIoTest.StatusIn.diStatusDachluftFeuchteMax	 := FALSE;
		END_IF

		//Modul 10 Luftgeschwindigkeit ****************************************************************************
		IF (cmModul10.StatusInput01.1 = FALSE AND cmModul10.StatusInput01.0 = TRUE) THEN
			hmiIoTest.StatusIn.diStatusLuftgeschwMin	:= TRUE;
		ELSE
			hmiIoTest.StatusIn.diStatusLuftgeschwMin	:= FALSE;
		END_IF
		IF (cmModul10.StatusInput01.1 = TRUE AND cmModul10.StatusInput01.0 = FALSE ) THEN
			hmiIoTest.StatusIn.diStatusLuftgeschwMax	:= TRUE;
		ELSE
			hmiIoTest.StatusIn.diStatusLuftgeschwMax	 := FALSE;
		END_IF
		IF ((cmModul10.StatusInput01.1 = TRUE AND cmModul10.StatusInput01.0 = TRUE) OR cmModul10.ai01 >= 32767) THEN
			hmiIoTest.StatusIn.diStatusLuftgeschwDrahtbruch := TRUE;
		ELSE
			hmiIoTest.StatusIn.diStatusLuftgeschwDrahtbruch := FALSE;
		END_IF

		//Modul 11 Differenzdruck ****************************************************************************
		IF (cmModul11.StatusInput01.1 = FALSE AND cmModul11.StatusInput01.0 = TRUE) THEN
			hmiIoTest.StatusIn.diStatusDifferenzdruckMin	:= TRUE;
		ELSE
			hmiIoTest.StatusIn.diStatusDifferenzdruckMin	:= FALSE;
		END_IF
		IF (cmModul11.StatusInput01.1 = TRUE AND cmModul11.StatusInput01.0 = FALSE ) THEN
			hmiIoTest.StatusIn.diStatusDifferenzdruckMax	 := TRUE;
		ELSE
			hmiIoTest.StatusIn.diStatusDifferenzdruckMax	 := FALSE;
		END_IF

	END_IF

	//============================================================================================================================================================================
	//Modulüberwachungen
	//============================================================================================================================================================================

	loc_Erforderl_Mod1	:= TRUE;
	loc_Erforderl_Mod2	:= TRUE;
	loc_Erforderl_Mod3	:= Aktoren.VentUndKlappen.Boxenklappe1Vorhanden OR Aktoren.VentUndKlappen.Boxenklappe2Vorhanden OR
		Betriebsparameter.Ausstattung.SensorFrischluft OR Betriebsparameter.Ausstattung.WarmluftofenTempVorgabe;
	loc_Erforderl_Mod4	:= TRUE;
	loc_Erforderl_Mod5	:= Betriebsparameter.Ausstattung.Warmluftofen OR Betriebsparameter.Ausstattung.Scheitholzofen OR Betriebsparameter.Ausstattung.Heizregister OR
		Betriebsparameter.Ausstattung.SensorTrockenluft;
	loc_Erforderl_Mod6	:= Aktoren.VentUndKlappen.Boxenklappe3Vorhanden OR Aktoren.VentUndKlappen.Boxenklappe4Vorhanden OR Betriebsparameter.Ausstattung.SensorAbluft;
	loc_Erforderl_Mod7	:= Betriebsparameter.Ausstattung.SensorAbluft;
	loc_Erforderl_Mod8	:= Betriebsparameter.Ausstattung.Abluftventilator OR Betriebsparameter.Ausstattung.Brandschutzklappe OR Betriebsparameter.Ausstattung.SensorDachluft;
	loc_Erforderl_Mod9	:= Betriebsparameter.Ausstattung.Abluftklappe OR Betriebsparameter.Ausstattung.SensorDachluft;
	loc_Erforderl_Mod10	:= Betriebsparameter.Ausstattung.Umschaltklappe1 OR Betriebsparameter.Ausstattung.Umschaltklappe2 OR
		Betriebsparameter.Ausstattung.SensorLuftgeschwindigkeit;
	loc_Erforderl_Mod11	:= Betriebsparameter.Ausstattung.Notstromaggregat OR Betriebsparameter.Ausstattung.SensorKanaldruck;
	loc_Erforderl_Mod12	:= Betriebsparameter.Ausstattung.Energiemessung;

	fbLascoFehl_0.FehlerIn	:= (loc_Erforderl_Mod1 AND NOT brModul01.ModulOk) OR (loc_Erforderl_Mod2 AND NOT cmModul02.ModulOk) OR
	(loc_Erforderl_Mod3 AND NOT cmModul03.ModulOk) OR (loc_Erforderl_Mod4 AND NOT cmModul04.ModulOk) OR (loc_Erforderl_Mod5 AND NOT cmModul05.ModulOk) OR
	(loc_Erforderl_Mod6 AND NOT cmModul06.ModulOk) OR (loc_Erforderl_Mod7 AND NOT cmModul07.ModulOk) OR (loc_Erforderl_Mod8 AND NOT cmModul08.ModulOk) OR
	(loc_Erforderl_Mod9 AND NOT cmModul09.ModulOk) OR (loc_Erforderl_Mod10 AND NOT cmModul10.ModulOk) OR (loc_Erforderl_Mod11 AND NOT cmModul11.ModulOk) OR
	(loc_Erforderl_Mod12 AND NOT gEnergiemessungModulOk);
	fbLascoFehl_0.Mode		:= 2;
	fbLascoFehl_0.Quit		:= hmiButtons.QuitFehler;
	fbLascoFehl_0.Tick		:= sekTick;
	fbLascoFehl_0();

	alarmSystem[FEHLER_KOMMUNIKATION_DISPLAY_IO] := fbLascoFehl_0.FehlerOut;

END_PROGRAM

PROGRAM _EXIT

END_PROGRAM
```

#### Variables.var - Local variables
```iecst
(*==========================================================================================================================================================*)
(*============================================ LOKALE VARIABLEN ============================================================================================*)
VAR
	sekTick : BOOL;
END_VAR
(*==========================================================================================================================================================*)
(*============================================ MODULE ======================================================================================================*)
VAR
	brModul01 : modBR7300;
	cmModul02 : modCM8281;
	cmModul03 : modCM8281;
	cmModul04 : modCM8281;
	cmModul05 : modCM8281;
	cmModul06 : modCM8281;
	cmModul07 : modCM8281;
	cmModul08 : modCM8281;
	cmModul09 : modCM8281;
	cmModul10 : modCM8281;
	cmModul11 : modCM8281;
END_VAR
(*==========================================================================================================================================================*)
(*============================================ FUNKTIONSBAUSTEINE =========================================================================================*)
VAR
	fbLascoZdxx_0 : fbLascoZdxx;
	LCRMovAvgFlt_0 : LCRMovAvgFlt;
	LCRMovAvgFlt_1 : LCRMovAvgFlt;
	LCRMovAvgFlt_2 : LCRMovAvgFlt;
	LCRMovAvgFlt_3 : LCRMovAvgFlt;
	LCRMovAvgFlt_4 : LCRMovAvgFlt;
	LCRMovAvgFlt_5 : LCRMovAvgFlt;
	LCRMovAvgFlt_6 : LCRMovAvgFlt;
	LCRMovAvgFlt_7 : LCRMovAvgFlt;
	LCRMovAvgFlt_8 : LCRMovAvgFlt;
	LCRMovAvgFlt_9 : LCRMovAvgFlt;
	LCRLimScal_0 : LCRLimScal;
	loc_Erforderl_Mod1 : BOOL;
	loc_Erforderl_Mod2 : BOOL;
	loc_Erforderl_Mod3 : BOOL;
	loc_Erforderl_Mod4 : BOOL;
	loc_Erforderl_Mod5 : BOOL;
	loc_Erforderl_Mod6 : BOOL;
	loc_Erforderl_Mod7 : BOOL;
	loc_Erforderl_Mod8 : BOOL;
	loc_Erforderl_Mod9 : BOOL;
	loc_Erforderl_Mod10 : BOOL;
	loc_Erforderl_Mod11 : BOOL;
	loc_Erforderl_Mod12 : BOOL;
	fbLascoFehl_0 : {REDUND_UNREPLICABLE} fbLascoFehl;
END_VAR
```

### Package Logical/Berechnung - Berechnung

### Berechnungen.var - Paket Variablen
```iecst
(*============================================================================================================================================*)
(*======================================== FUNKTIONSBAUSTEINE FÜR FÜHLERBERECHNUNGEN ====================================================*)
VAR
	fbSchlechtwetterBox1 : {REDUND_UNREPLICABLE} fbCControlWitterung;
	fbSchlechtwetterBox2 : {REDUND_UNREPLICABLE} fbCControlWitterung;
	fbSchlechtwetterBox3 : {REDUND_UNREPLICABLE} fbCControlWitterung;
	fbSchlechtwetterBox4 : {REDUND_UNREPLICABLE} fbCControlWitterung;
	fbSchlechtwetterBox5 : {REDUND_UNREPLICABLE} fbCControlWitterung;
	fbSchlechtwetterBox6 : {REDUND_UNREPLICABLE} fbCControlWitterung;
	Frischluftsensor : {REDUND_UNREPLICABLE} fbMathLuft;
	Dachluftsensor : {REDUND_UNREPLICABLE} fbMathLuft;
	Trockenluftsensor : {REDUND_UNREPLICABLE} fbMathLuft;
	Abluftsensor : {REDUND_UNREPLICABLE} fbMathLuft;
	Drucksensor : {REDUND_UNREPLICABLE} fbMathTrLftDruck;
END_VAR
```

### Program Logical/Berechnung/Berechnung (IEC) - Berechnungen aus Fühlerwerten

#### Berechnung.st - Zyklischer Code
```iecst
PROGRAM _CYCLIC

	//====================================================================================================================================================
	//Berechnungen aus Fühlerwerten
	//====================================================================================================================================================

	//Berechnungen Frischluftsensor
	//*****************************
	Frischluftsensor.Freigabe							:= Betriebsparameter.Ausstattung.SensorFrischluft AND NOT alarmFehler[FEHLER_SENSOR_FRISCHLUFT];
	Frischluftsensor.LuftTemperatur						:= aiFrischluftTemperatur;
	Frischluftsensor.LuftRelFeuchte						:= aiFrischluftFeuchte;
	Frischluftsensor.MeterUeberAdria					:= Betriebsparameter.Allgemein.StandortHoehe;
	Frischluftsensor();

	gStatusAnlage.Berechnungen.FrischluftSattDefizit	:= Frischluftsensor.LuftSaettigungsdefizit;

	//Berechnungen Trockenluftsensor
	//******************************
	Trockenluftsensor.Freigabe							:= Betriebsparameter.Ausstattung.SensorTrockenluft AND NOT alarmFehler[FEHLER_SENSOR_TROCKENLUFT];
	Trockenluftsensor.LuftTemperatur					:= aiTrockenluftTemperatur;
	Trockenluftsensor.LuftRelFeuchte					:= aiTrockenluftFeuchte;
	Trockenluftsensor.MeterUeberAdria					:= Betriebsparameter.Allgemein.StandortHoehe;
	Trockenluftsensor();

	gStatusAnlage.Berechnungen.TrockenluftSattDefizit	:= Trockenluftsensor.LuftSaettigungsdefizit;

	//Berechnungen Dachluftsensor
	//******************************
	Dachluftsensor.Freigabe							:= Betriebsparameter.Ausstattung.SensorDachluft AND NOT alarmFehler[FEHLER_SENSOR_DACHLUFT];
	Dachluftsensor.LuftTemperatur					:= aiDachluftTemperatur;
	Dachluftsensor.LuftRelFeuchte					:= aiDachluftFeuchte;
	Dachluftsensor.MeterUeberAdria					:= Betriebsparameter.Allgemein.StandortHoehe;
	Dachluftsensor();

	gStatusAnlage.Berechnungen.DachluftSattDefizit	:= Dachluftsensor.LuftSaettigungsdefizit;

	//Berechnungen Abluftsensor
	//************************
	Abluftsensor.Freigabe							:= Betriebsparameter.Ausstattung.SensorAbluft AND NOT alarmFehler[FEHLER_SENSOR_ABLUFT];
	Abluftsensor.LuftTemperatur						:= aiAbluftTemperatur;
	Abluftsensor.LuftRelFeuchte						:= aiAbluftFeuchte;
	Abluftsensor.MeterUeberAdria					:= Betriebsparameter.Allgemein.StandortHoehe;
	Abluftsensor();

	gStatusAnlage.Berechnungen.AbluftSattDefizit	:= Abluftsensor.LuftSaettigungsdefizit;

	//Berechnungen Drucksensor
	//************************
	Drucksensor.Freigabe						:= (doVentilator1Ein OR doVentilator2Ein) AND Betriebsparameter.Ausstattung.SensorKanaldruck AND NOT alarmFehler[FEHLER_SENSOR_KANALDRUCK];
	Drucksensor.TrockenluftDruck				:= aiDifferenzdruck;
	Drucksensor();

	IF doVentilator1Ein OR doVentilator2Ein THEN
		gStatusAnlage.Berechnungen.Kanaldruck_mmWs	:= Drucksensor.LuftDruck_mmWS;
	ELSE
		gStatusAnlage.Berechnungen.Kanaldruck_mmWs	:= 0.0;
	END_IF

	//====================================================================================================================================================
	//Bestimmung der Witterungsverhältnisse
	//====================================================================================================================================================

	//Variable "Wetter is Schlecht" generieren, wenn eine der eingeschalteten Boxen schlechte Witterung ausgibt
	gStatusAnlage.WetterIstSchlecht := (Boxen.Box1In.WetterIstSchlecht AND Boxen.Box1Out.BoxBereit) OR (Boxen.Box2In.WetterIstSchlecht AND Boxen.Box2Out.BoxBereit) OR
	(Boxen.Box3In.WetterIstSchlecht AND Boxen.Box3Out.BoxBereit) OR (Boxen.Box4In.WetterIstSchlecht AND Boxen.Box4Out.BoxBereit) OR
	(Boxen.Box5In.WetterIstSchlecht AND Boxen.Box5Out.BoxBereit) OR (Boxen.Box6In.WetterIstSchlecht AND Boxen.Box6Out.BoxBereit);

	//Box 1	**********************************************************************************************************************************************
	fbSchlechtwetterBox1.Freigabe						:= TRUE;
	fbSchlechtwetterBox1.AuswahlSensor					:= Betriebsparameter.SchlechtwetterBoxen[1].AuswahlSensorGrenzwert;
	fbSchlechtwetterBox1.FrischluftSaettigungsdefizit	:= gStatusAnlage.Berechnungen.FrischluftSattDefizit;
	fbSchlechtwetterBox1.DachluftSaettigungsdefizit		:= gStatusAnlage.Berechnungen.DachluftSattDefizit;
	fbSchlechtwetterBox1.TrockenluftSaettigungsdefizit	:= gStatusAnlage.Berechnungen.TrockenluftSattDefizit;
	fbSchlechtwetterBox1.SensorFrischluftVhd			:= Betriebsparameter.Ausstattung.SensorFrischluft AND NOT alarmFehler[FEHLER_SENSOR_FRISCHLUFT];
	fbSchlechtwetterBox1.SensorDachluftVhd				:= Betriebsparameter.Ausstattung.SensorDachluft AND NOT alarmFehler[FEHLER_SENSOR_DACHLUFT];
	fbSchlechtwetterBox1.SensorTrockenluftVhd			:= Betriebsparameter.Ausstattung.SensorTrockenluft AND NOT alarmFehler[FEHLER_SENSOR_TROCKENLUFT];
	fbSchlechtwetterBox1.VerzWetterwechsel				:= Betriebsparameter.Schrittkette.VerzWetterwechsel;

	fbSchlechtwetterBox1.MaterialfeuchteStufe[1]		:= Betriebsparameter.SchlechtwetterBoxen[1].Stufe[1].MaterialfeuchteStufe;
	fbSchlechtwetterBox1.MaterialfeuchteStufe[2]		:= Betriebsparameter.SchlechtwetterBoxen[1].Stufe[2].MaterialfeuchteStufe;
	fbSchlechtwetterBox1.MaterialfeuchteStufe[3]		:= Betriebsparameter.SchlechtwetterBoxen[1].Stufe[3].MaterialfeuchteStufe;
	fbSchlechtwetterBox1.MaterialfeuchteStufe[4]		:= Betriebsparameter.SchlechtwetterBoxen[1].Stufe[4].MaterialfeuchteStufe;
	fbSchlechtwetterBox1.MaterialfeuchteStufe[5]		:= Betriebsparameter.SchlechtwetterBoxen[1].Stufe[5].MaterialfeuchteStufe;
	fbSchlechtwetterBox1.MaterialfeuchteStufe[6]		:= Betriebsparameter.SchlechtwetterBoxen[1].Stufe[6].MaterialfeuchteStufe;

	fbSchlechtwetterBox1.GrenzwertStufeAktuell			:= Betriebsparameter.SchlechtwetterBoxen[1].Stufe[fbSchlechtwetterBox1.StufeAktuell].Saettigungsdefizit;
	fbSchlechtwetterBox1.HystereseGrenzwert				:= Betriebsparameter.SchlechtwetterBoxen[1].HystereseGrenzwert;
	fbSchlechtwetterBox1.MaterialfeuchteIst				:= Betriebsparameter.SchlechtwetterBoxen[1].MaterialfeuchteIst;

	fbSchlechtwetterBox1.SchlechtwetterPausezeitStufe[fbSchlechtwetterBox1.StufeAktuell] :=
	Betriebsparameter.SchlechtwetterBoxen[1].Stufe[fbSchlechtwetterBox1.StufeAktuell].SchlechtwetterZeitPause;
	fbSchlechtwetterBox1.SchlechtwetterPulszeitStufe[fbSchlechtwetterBox1.StufeAktuell] :=
	Betriebsparameter.SchlechtwetterBoxen[1].Stufe[fbSchlechtwetterBox1.StufeAktuell].SchlechtwetterZeitLauf;

	//Box 2	**********************************************************************************************************************************************
	fbSchlechtwetterBox2.Freigabe						:= TRUE;
	fbSchlechtwetterBox2.AuswahlSensor					:= Betriebsparameter.SchlechtwetterBoxen[2].AuswahlSensorGrenzwert;
	fbSchlechtwetterBox2.FrischluftSaettigungsdefizit	:= gStatusAnlage.Berechnungen.FrischluftSattDefizit;
	fbSchlechtwetterBox2.DachluftSaettigungsdefizit		:= gStatusAnlage.Berechnungen.DachluftSattDefizit;
	fbSchlechtwetterBox2.TrockenluftSaettigungsdefizit	:= gStatusAnlage.Berechnungen.TrockenluftSattDefizit;
	fbSchlechtwetterBox2.SensorFrischluftVhd			:= Betriebsparameter.Ausstattung.SensorFrischluft AND NOT alarmFehler[FEHLER_SENSOR_FRISCHLUFT];
	fbSchlechtwetterBox2.SensorDachluftVhd				:= Betriebsparameter.Ausstattung.SensorDachluft AND NOT alarmFehler[FEHLER_SENSOR_DACHLUFT];
	fbSchlechtwetterBox2.SensorTrockenluftVhd			:= Betriebsparameter.Ausstattung.SensorTrockenluft AND NOT alarmFehler[FEHLER_SENSOR_TROCKENLUFT];
	fbSchlechtwetterBox2.VerzWetterwechsel				:= Betriebsparameter.Schrittkette.VerzWetterwechsel;

	fbSchlechtwetterBox2.MaterialfeuchteStufe[1]		:= Betriebsparameter.SchlechtwetterBoxen[2].Stufe[1].MaterialfeuchteStufe;
	fbSchlechtwetterBox2.MaterialfeuchteStufe[2]		:= Betriebsparameter.SchlechtwetterBoxen[2].Stufe[2].MaterialfeuchteStufe;
	fbSchlechtwetterBox2.MaterialfeuchteStufe[3]		:= Betriebsparameter.SchlechtwetterBoxen[2].Stufe[3].MaterialfeuchteStufe;
	fbSchlechtwetterBox2.MaterialfeuchteStufe[4]		:= Betriebsparameter.SchlechtwetterBoxen[2].Stufe[4].MaterialfeuchteStufe;
	fbSchlechtwetterBox2.MaterialfeuchteStufe[5]		:= Betriebsparameter.SchlechtwetterBoxen[2].Stufe[5].MaterialfeuchteStufe;
	fbSchlechtwetterBox2.MaterialfeuchteStufe[6]		:= Betriebsparameter.SchlechtwetterBoxen[2].Stufe[6].MaterialfeuchteStufe;

	fbSchlechtwetterBox2.GrenzwertStufeAktuell			:= Betriebsparameter.SchlechtwetterBoxen[2].Stufe[fbSchlechtwetterBox2.StufeAktuell].Saettigungsdefizit;
	fbSchlechtwetterBox2.HystereseGrenzwert				:= Betriebsparameter.SchlechtwetterBoxen[1].HystereseGrenzwert; //Gleiche Hysterese für alle Boxen
	fbSchlechtwetterBox2.MaterialfeuchteIst				:= Betriebsparameter.SchlechtwetterBoxen[2].MaterialfeuchteIst;

	fbSchlechtwetterBox2.SchlechtwetterPausezeitStufe[fbSchlechtwetterBox2.StufeAktuell] :=
	Betriebsparameter.SchlechtwetterBoxen[2].Stufe[fbSchlechtwetterBox2.StufeAktuell].SchlechtwetterZeitPause;
	fbSchlechtwetterBox2.SchlechtwetterPulszeitStufe[fbSchlechtwetterBox2.StufeAktuell] :=
	Betriebsparameter.SchlechtwetterBoxen[2].Stufe[fbSchlechtwetterBox2.StufeAktuell].SchlechtwetterZeitLauf;

	//Box 3	**********************************************************************************************************************************************
	fbSchlechtwetterBox3.Freigabe						:= TRUE;
	fbSchlechtwetterBox3.AuswahlSensor					:= Betriebsparameter.SchlechtwetterBoxen[3].AuswahlSensorGrenzwert;
	fbSchlechtwetterBox3.FrischluftSaettigungsdefizit	:= gStatusAnlage.Berechnungen.FrischluftSattDefizit;
	fbSchlechtwetterBox3.DachluftSaettigungsdefizit		:= gStatusAnlage.Berechnungen.DachluftSattDefizit;
	fbSchlechtwetterBox3.TrockenluftSaettigungsdefizit	:= gStatusAnlage.Berechnungen.TrockenluftSattDefizit;
	fbSchlechtwetterBox3.SensorFrischluftVhd			:= Betriebsparameter.Ausstattung.SensorFrischluft AND NOT alarmFehler[FEHLER_SENSOR_FRISCHLUFT];
	fbSchlechtwetterBox3.SensorDachluftVhd				:= Betriebsparameter.Ausstattung.SensorDachluft AND NOT alarmFehler[FEHLER_SENSOR_DACHLUFT];
	fbSchlechtwetterBox3.SensorTrockenluftVhd			:= Betriebsparameter.Ausstattung.SensorTrockenluft AND NOT alarmFehler[FEHLER_SENSOR_TROCKENLUFT];
	fbSchlechtwetterBox3.VerzWetterwechsel				:= Betriebsparameter.Schrittkette.VerzWetterwechsel;

	fbSchlechtwetterBox3.MaterialfeuchteStufe[1]		:= Betriebsparameter.SchlechtwetterBoxen[3].Stufe[1].MaterialfeuchteStufe;
	fbSchlechtwetterBox3.MaterialfeuchteStufe[2]		:= Betriebsparameter.SchlechtwetterBoxen[3].Stufe[2].MaterialfeuchteStufe;
	fbSchlechtwetterBox3.MaterialfeuchteStufe[3]		:= Betriebsparameter.SchlechtwetterBoxen[3].Stufe[3].MaterialfeuchteStufe;
	fbSchlechtwetterBox3.MaterialfeuchteStufe[4]		:= Betriebsparameter.SchlechtwetterBoxen[3].Stufe[4].MaterialfeuchteStufe;
	fbSchlechtwetterBox3.MaterialfeuchteStufe[5]		:= Betriebsparameter.SchlechtwetterBoxen[3].Stufe[5].MaterialfeuchteStufe;
	fbSchlechtwetterBox3.MaterialfeuchteStufe[6]		:= Betriebsparameter.SchlechtwetterBoxen[3].Stufe[6].MaterialfeuchteStufe;

	fbSchlechtwetterBox3.GrenzwertStufeAktuell			:= Betriebsparameter.SchlechtwetterBoxen[3].Stufe[fbSchlechtwetterBox3.StufeAktuell].Saettigungsdefizit;
	fbSchlechtwetterBox3.HystereseGrenzwert				:= Betriebsparameter.SchlechtwetterBoxen[1].HystereseGrenzwert; //Gleiche Hysterese für alle Boxen
	fbSchlechtwetterBox3.MaterialfeuchteIst				:= Betriebsparameter.SchlechtwetterBoxen[3].MaterialfeuchteIst;

	fbSchlechtwetterBox3.SchlechtwetterPausezeitStufe[fbSchlechtwetterBox3.StufeAktuell] :=
	Betriebsparameter.SchlechtwetterBoxen[3].Stufe[fbSchlechtwetterBox3.StufeAktuell].SchlechtwetterZeitPause;
	fbSchlechtwetterBox3.SchlechtwetterPulszeitStufe[fbSchlechtwetterBox3.StufeAktuell] :=
	Betriebsparameter.SchlechtwetterBoxen[3].Stufe[fbSchlechtwetterBox3.StufeAktuell].SchlechtwetterZeitLauf;

	//Box 4	**********************************************************************************************************************************************
	fbSchlechtwetterBox4.Freigabe						:= TRUE;
	fbSchlechtwetterBox4.AuswahlSensor					:= Betriebsparameter.SchlechtwetterBoxen[4].AuswahlSensorGrenzwert;
	fbSchlechtwetterBox4.FrischluftSaettigungsdefizit	:= gStatusAnlage.Berechnungen.FrischluftSattDefizit;
	fbSchlechtwetterBox4.DachluftSaettigungsdefizit		:= gStatusAnlage.Berechnungen.DachluftSattDefizit;
	fbSchlechtwetterBox4.TrockenluftSaettigungsdefizit	:= gStatusAnlage.Berechnungen.TrockenluftSattDefizit;
	fbSchlechtwetterBox4.SensorFrischluftVhd			:= Betriebsparameter.Ausstattung.SensorFrischluft AND NOT alarmFehler[FEHLER_SENSOR_FRISCHLUFT];
	fbSchlechtwetterBox4.SensorDachluftVhd				:= Betriebsparameter.Ausstattung.SensorDachluft AND NOT alarmFehler[FEHLER_SENSOR_DACHLUFT];
	fbSchlechtwetterBox4.SensorTrockenluftVhd			:= Betriebsparameter.Ausstattung.SensorTrockenluft AND NOT alarmFehler[FEHLER_SENSOR_TROCKENLUFT];
	fbSchlechtwetterBox4.VerzWetterwechsel				:= Betriebsparameter.Schrittkette.VerzWetterwechsel;

	fbSchlechtwetterBox4.MaterialfeuchteStufe[1]		:= Betriebsparameter.SchlechtwetterBoxen[4].Stufe[1].MaterialfeuchteStufe;
	fbSchlechtwetterBox4.MaterialfeuchteStufe[2]		:= Betriebsparameter.SchlechtwetterBoxen[4].Stufe[2].MaterialfeuchteStufe;
	fbSchlechtwetterBox4.MaterialfeuchteStufe[3]		:= Betriebsparameter.SchlechtwetterBoxen[4].Stufe[3].MaterialfeuchteStufe;
	fbSchlechtwetterBox4.MaterialfeuchteStufe[4]		:= Betriebsparameter.SchlechtwetterBoxen[4].Stufe[4].MaterialfeuchteStufe;
	fbSchlechtwetterBox4.MaterialfeuchteStufe[5]		:= Betriebsparameter.SchlechtwetterBoxen[4].Stufe[5].MaterialfeuchteStufe;
	fbSchlechtwetterBox4.MaterialfeuchteStufe[6]		:= Betriebsparameter.SchlechtwetterBoxen[4].Stufe[6].MaterialfeuchteStufe;

	fbSchlechtwetterBox4.GrenzwertStufeAktuell			:= Betriebsparameter.SchlechtwetterBoxen[4].Stufe[fbSchlechtwetterBox4.StufeAktuell].Saettigungsdefizit;
	fbSchlechtwetterBox4.HystereseGrenzwert				:= Betriebsparameter.SchlechtwetterBoxen[1].HystereseGrenzwert; //Gleiche Hysterese für alle Boxen
	fbSchlechtwetterBox4.MaterialfeuchteIst				:= Betriebsparameter.SchlechtwetterBoxen[4].MaterialfeuchteIst;

	fbSchlechtwetterBox4.SchlechtwetterPausezeitStufe[fbSchlechtwetterBox4.StufeAktuell] :=
	Betriebsparameter.SchlechtwetterBoxen[4].Stufe[fbSchlechtwetterBox4.StufeAktuell].SchlechtwetterZeitPause;
	fbSchlechtwetterBox4.SchlechtwetterPulszeitStufe[fbSchlechtwetterBox4.StufeAktuell] :=
	Betriebsparameter.SchlechtwetterBoxen[4].Stufe[fbSchlechtwetterBox4.StufeAktuell].SchlechtwetterZeitLauf;

	//Box 5	**********************************************************************************************************************************************
	fbSchlechtwetterBox5.Freigabe						:= TRUE;
	fbSchlechtwetterBox5.AuswahlSensor					:= Betriebsparameter.SchlechtwetterBoxen[5].AuswahlSensorGrenzwert;
	fbSchlechtwetterBox5.FrischluftSaettigungsdefizit	:= gStatusAnlage.Berechnungen.FrischluftSattDefizit;
	fbSchlechtwetterBox5.DachluftSaettigungsdefizit		:= gStatusAnlage.Berechnungen.DachluftSattDefizit;
	fbSchlechtwetterBox5.TrockenluftSaettigungsdefizit	:= gStatusAnlage.Berechnungen.TrockenluftSattDefizit;
	fbSchlechtwetterBox5.SensorFrischluftVhd			:= Betriebsparameter.Ausstattung.SensorFrischluft AND NOT alarmFehler[FEHLER_SENSOR_FRISCHLUFT];
	fbSchlechtwetterBox5.SensorDachluftVhd				:= Betriebsparameter.Ausstattung.SensorDachluft AND NOT alarmFehler[FEHLER_SENSOR_DACHLUFT];
	fbSchlechtwetterBox5.SensorTrockenluftVhd			:= Betriebsparameter.Ausstattung.SensorTrockenluft AND NOT alarmFehler[FEHLER_SENSOR_TROCKENLUFT];
	fbSchlechtwetterBox5.VerzWetterwechsel				:= Betriebsparameter.Schrittkette.VerzWetterwechsel;

	fbSchlechtwetterBox5.MaterialfeuchteStufe[1]		:= Betriebsparameter.SchlechtwetterBoxen[5].Stufe[1].MaterialfeuchteStufe;
	fbSchlechtwetterBox5.MaterialfeuchteStufe[2]		:= Betriebsparameter.SchlechtwetterBoxen[5].Stufe[2].MaterialfeuchteStufe;
	fbSchlechtwetterBox5.MaterialfeuchteStufe[3]		:= Betriebsparameter.SchlechtwetterBoxen[5].Stufe[3].MaterialfeuchteStufe;
	fbSchlechtwetterBox5.MaterialfeuchteStufe[4]		:= Betriebsparameter.SchlechtwetterBoxen[5].Stufe[4].MaterialfeuchteStufe;
	fbSchlechtwetterBox5.MaterialfeuchteStufe[5]		:= Betriebsparameter.SchlechtwetterBoxen[5].Stufe[5].MaterialfeuchteStufe;
	fbSchlechtwetterBox5.MaterialfeuchteStufe[6]		:= Betriebsparameter.SchlechtwetterBoxen[5].Stufe[6].MaterialfeuchteStufe;

	fbSchlechtwetterBox5.GrenzwertStufeAktuell			:= Betriebsparameter.SchlechtwetterBoxen[5].Stufe[fbSchlechtwetterBox5.StufeAktuell].Saettigungsdefizit;
	fbSchlechtwetterBox5.HystereseGrenzwert				:= Betriebsparameter.SchlechtwetterBoxen[1].HystereseGrenzwert; //Gleiche Hysterese für alle Boxen
	fbSchlechtwetterBox5.MaterialfeuchteIst				:= Betriebsparameter.SchlechtwetterBoxen[5].MaterialfeuchteIst;

	fbSchlechtwetterBox5.SchlechtwetterPausezeitStufe[fbSchlechtwetterBox5.StufeAktuell] :=
	Betriebsparameter.SchlechtwetterBoxen[5].Stufe[fbSchlechtwetterBox5.StufeAktuell].SchlechtwetterZeitPause;
	fbSchlechtwetterBox5.SchlechtwetterPulszeitStufe[fbSchlechtwetterBox5.StufeAktuell] :=
	Betriebsparameter.SchlechtwetterBoxen[5].Stufe[fbSchlechtwetterBox5.StufeAktuell].SchlechtwetterZeitLauf;

	//Box 6	**********************************************************************************************************************************************
	fbSchlechtwetterBox6.Freigabe						:= TRUE;
	fbSchlechtwetterBox6.AuswahlSensor					:= Betriebsparameter.SchlechtwetterBoxen[6].AuswahlSensorGrenzwert;
	fbSchlechtwetterBox6.FrischluftSaettigungsdefizit	:= gStatusAnlage.Berechnungen.FrischluftSattDefizit;
	fbSchlechtwetterBox6.DachluftSaettigungsdefizit		:= gStatusAnlage.Berechnungen.DachluftSattDefizit;
	fbSchlechtwetterBox6.TrockenluftSaettigungsdefizit	:= gStatusAnlage.Berechnungen.TrockenluftSattDefizit;
	fbSchlechtwetterBox6.SensorFrischluftVhd			:= Betriebsparameter.Ausstattung.SensorFrischluft AND NOT alarmFehler[FEHLER_SENSOR_FRISCHLUFT];
	fbSchlechtwetterBox6.SensorDachluftVhd				:= Betriebsparameter.Ausstattung.SensorDachluft AND NOT alarmFehler[FEHLER_SENSOR_DACHLUFT];
	fbSchlechtwetterBox6.SensorTrockenluftVhd			:= Betriebsparameter.Ausstattung.SensorTrockenluft AND NOT alarmFehler[FEHLER_SENSOR_TROCKENLUFT];
	fbSchlechtwetterBox6.VerzWetterwechsel				:= Betriebsparameter.Schrittkette.VerzWetterwechsel;

	fbSchlechtwetterBox6.MaterialfeuchteStufe[1]		:= Betriebsparameter.SchlechtwetterBoxen[6].Stufe[1].MaterialfeuchteStufe;
	fbSchlechtwetterBox6.MaterialfeuchteStufe[2]		:= Betriebsparameter.SchlechtwetterBoxen[6].Stufe[2].MaterialfeuchteStufe;
	fbSchlechtwetterBox6.MaterialfeuchteStufe[3]		:= Betriebsparameter.SchlechtwetterBoxen[6].Stufe[3].MaterialfeuchteStufe;
	fbSchlechtwetterBox6.MaterialfeuchteStufe[4]		:= Betriebsparameter.SchlechtwetterBoxen[6].Stufe[4].MaterialfeuchteStufe;
	fbSchlechtwetterBox6.MaterialfeuchteStufe[5]		:= Betriebsparameter.SchlechtwetterBoxen[6].Stufe[5].MaterialfeuchteStufe;
	fbSchlechtwetterBox6.MaterialfeuchteStufe[6]		:= Betriebsparameter.SchlechtwetterBoxen[6].Stufe[6].MaterialfeuchteStufe;

	fbSchlechtwetterBox6.GrenzwertStufeAktuell			:= Betriebsparameter.SchlechtwetterBoxen[6].Stufe[fbSchlechtwetterBox6.StufeAktuell].Saettigungsdefizit;
	fbSchlechtwetterBox6.HystereseGrenzwert				:= Betriebsparameter.SchlechtwetterBoxen[1].HystereseGrenzwert; //Gleiche Hysterese für alle Boxen
	fbSchlechtwetterBox6.MaterialfeuchteIst				:= Betriebsparameter.SchlechtwetterBoxen[6].MaterialfeuchteIst;

	fbSchlechtwetterBox6.SchlechtwetterPausezeitStufe[fbSchlechtwetterBox6.StufeAktuell] :=
	Betriebsparameter.SchlechtwetterBoxen[6].Stufe[fbSchlechtwetterBox6.StufeAktuell].SchlechtwetterZeitPause;
	fbSchlechtwetterBox6.SchlechtwetterPulszeitStufe[fbSchlechtwetterBox6.StufeAktuell] :=
	Betriebsparameter.SchlechtwetterBoxen[6].Stufe[fbSchlechtwetterBox6.StufeAktuell].SchlechtwetterZeitLauf;

END_PROGRAM
```

### Package Logical/Alarmsystem - Fehler- und Warnungsgenerierung

### Program Logical/Alarmsystem/Alarm (IEC) - Alarmgenerierung

#### AlarmCyclic.st - Zyklischer Code
```iecst
PROGRAM _INIT

	init	:= FALSE;

END_PROGRAM

PROGRAM _CYCLIC

	//Sekundentick generieren
	//=======================
	eUhr(Freigabe:= TRUE);
	fbLascoZdxx_0(IN := eUhr.Sekunde);
	sekTick	:= fbLascoZdxx_0.Q;

	//Fehlergenerierung eingeschaltet *****************************************************************************************************************************************************************
	IF init THEN

		//=======================================================================================================================================================
		//FEHLER ------------------------------ FEHLER ------------------------------ FEHLER ------------------------------ FEHLER ------------------------------
		//=======================================================================================================================================================

		//00) Fehler Absicherung 24VDC
		alarmFehler[FEHLER_24VDC]			:= NOT di24VDCinternIstOk;

		//01) Fehler FU Kompressor Modul 1
		alarmFehler[FEHLER_FU_KOMPRESSOR_MODUL1]	:= Aktoren.KompressorModul1.StoerungOut;

		//02) Fehler FU Kompressor Modul 2
		alarmFehler[FEHLER_FU_KOMPRESSOR_MODUL2]	:= Aktoren.KompressorModul2.StoerungOut;

		//03) Fehler Betriebsmeldung Kompressor Modul 1
		fbLascoFehl_0(FehlerIn := doKompressorEinModul1 AND NOT diBetriebsmldgKompressorModul1,
		VerzZeit := Betriebsparameter.Allgemein.VerzoegerungFehler, Quit := hmiButtons.QuitFehler, Tick := sekTick, Mode := 1);
		alarmFehler[FEHLER_BETRIEBSMLDG_KOMPR_MOD1]	:= fbLascoFehl_0.FehlerOut;

		//04) Fehler Betriebsmeldung Kompressor Modul 2
		fbLascoFehl_1(FehlerIn := gModul2Vorhanden AND doKompressorEinModul2 AND NOT diBetriebsmldgKompressorModul2,
		VerzZeit := Betriebsparameter.Allgemein.VerzoegerungFehler, Quit := hmiButtons.QuitFehler, Tick := sekTick, Mode := 1);
		alarmFehler[FEHLER_BETRIEBSMLDG_KOMPR_MOD2]	:= fbLascoFehl_1.FehlerOut;

		//05) Fehler Betriebsmeldung Ventilator 1
		fbLascoFehl_2(FehlerIn := Aktoren.VentUndKlappen.FehlerFuVentilator1,
		VerzZeit := 0, Quit := hmiButtons.QuitFehler, Tick := sekTick, Mode := 1);
		alarmFehler[FEHLER_BETRIEBSMLDG_VENTILATOR1]	:= fbLascoFehl_2.FehlerOut;

		//06) Fehler Betriebsmeldung Ventilator 2
		fbLascoFehl_3(FehlerIn := Aktoren.VentUndKlappen.FehlerFuVentilator2,
		VerzZeit := 0, Quit := hmiButtons.QuitFehler, Tick := sekTick, Mode := 1);
		alarmFehler[FEHLER_BETRIEBSMLDG_VENTILATOR2]	:= fbLascoFehl_3.FehlerOut;

		//07) Fehler Betriebsmeldung Abluftventilator
		fbLascoFehl_4(FehlerIn := Aktoren.Abluftventilator.FehlerOut,
		VerzZeit := 0, Quit := hmiButtons.QuitFehler, Tick := sekTick, Mode := 1);
		alarmFehler[FEHLER_BETRIEBSMLDG_ABLUFTVENT]	:= fbLascoFehl_4.FehlerOut;

		//08) Fehler Hochdruck Modul 1
		fbLascoFehl_5(FehlerIn :=  Betriebsparameter.Ausstattung.Entfeuchter AND NOT diHochdruckOkModul1, VerzZeit := 0,
		Quit := hmiButtons.QuitFehler, Tick := sekTick, Mode := 0);
		alarmFehler[FEHLER_HOCHDRUCK_MODUL1]			:= fbLascoFehl_5.FehlerOut;

		//09) Fehler Hochdruck Modul 2
		fbLascoFehl_6(FehlerIn :=  Betriebsparameter.Ausstattung.Entfeuchter AND gModul2Vorhanden AND NOT diHochdruckOkModul2, VerzZeit := 0,
		Quit := hmiButtons.QuitFehler, Tick := sekTick, Mode := 0);
		alarmFehler[FEHLER_HOCHDRUCK_MODUL2]			:= fbLascoFehl_6.FehlerOut;

		//10) Fehler Niederdruck Modul 1
		fbLascoFehl_7(FehlerIn := Betriebsparameter.Ausstattung.Entfeuchter AND NOT diNiederdruckOkModul1, VerzZeit := 0,
		Quit := hmiButtons.QuitFehler, Tick := sekTick, Mode := 0);
		alarmFehler[FEHLER_NIEDERDRUCK_MODUL1]			:= fbLascoFehl_7.FehlerOut;

		//11) Fehler Niederdruck Modul 2
		fbLascoFehl_8(FehlerIn := Betriebsparameter.Ausstattung.Entfeuchter AND gModul2Vorhanden AND NOT diNiederdruckOkModul2,
		VerzZeit := 0, Quit := hmiButtons.QuitFehler, Tick := sekTick, Mode := 0);
		alarmFehler[FEHLER_NIEDERDRUCK_MODUL2]			:= fbLascoFehl_8.FehlerOut;

		//12) Fehler Öldruck Kompressor Modul 1
		fbLascoFehl_9(FehlerIn := Betriebsparameter.Ausstattung.Entfeuchter AND NOT diOeldruckKompressorModul1,
		VerzZeit := 0, Quit := hmiButtons.QuitFehler, Tick := sekTick, Mode := 0);
		alarmFehler[FEHLER_OELDRUCK_KOMPR_MOD1]			:= fbLascoFehl_9.FehlerOut;

		//13) Fehler Öldruck Kompressor Modul 2
		fbLascoFehl_10(FehlerIn := Betriebsparameter.Ausstattung.Entfeuchter AND gModul2Vorhanden AND NOT diOeldruckKompressorModul2,
		VerzZeit := 0, Quit := hmiButtons.QuitFehler, Tick := sekTick, Mode := 0);
		alarmFehler[FEHLER_OELDRUCK_KOMPR_MOD2]			:= fbLascoFehl_10.FehlerOut;

		//14) Fehler Kopftemperatur Kompressor Modul 1
		fbLascoFehl_11(FehlerIn := Betriebsparameter.Ausstattung.Entfeuchter AND NOT diKopftempKompressorModul1,
		VerzZeit := 0, Quit := hmiButtons.QuitFehler, Tick := sekTick, Mode := 0);
		alarmFehler[FEHLER_KOPFTEMP_KOMPR_MOD1]			:= fbLascoFehl_11.FehlerOut;

		//15) Fehler Kopftemperatur Kompressor Modul 2
		fbLascoFehl_12(FehlerIn := Betriebsparameter.Ausstattung.Entfeuchter AND gModul2Vorhanden AND NOT diKopftempKompressorModul2,
		VerzZeit := 0, Quit := hmiButtons.QuitFehler, Tick := sekTick, Mode := 0);
		alarmFehler[FEHLER_KOPFTEMP_KOMPR_MOD2]			:= fbLascoFehl_12.FehlerOut;

		//16) Fehler Vollschutz Kompressor Modul 1
		fbLascoFehl_13(FehlerIn := Betriebsparameter.Ausstattung.Entfeuchter AND NOT diVollschutzKompressorModul1,
		VerzZeit := 0, Quit := hmiButtons.QuitFehler, Tick := sekTick, Mode := 0);
		alarmFehler[FEHLER_VOLLSCHUTZ_KOMPR_MOD1]			:= fbLascoFehl_13.FehlerOut;

		//17) Fehler Vollschutz Kompressor Modul 2
		fbLascoFehl_14(FehlerIn := Betriebsparameter.Ausstattung.Entfeuchter AND gModul2Vorhanden AND NOT diVollschutzKompressorModul2,
		VerzZeit := 0, Quit := hmiButtons.QuitFehler, Tick := sekTick, Mode := 0);
		alarmFehler[FEHLER_VOLLSCHUTZ_KOMPR_MOD2]			:= fbLascoFehl_14.FehlerOut;

		//18) Fehler Betriebsmeldung Warmluftofen
		alarmFehler[FEHLER_BETRIEBSMLDG_WARMLUFTOFEN]	:= Aktoren.Warmluftofen.FehlerBetriebsmeldungOut;

		//19) Fehler Betriebsmeldung Notstromaggregat
		alarmFehler[FEHLER_BETRIEBSMLDG_NOTSTROM]		:= Aktoren.Notstromaggregat.FehlerOut;

		//20 - 31) Sensoren
		fbLascoFehl_15(FehlerIn := ((*diStatusFrischluftFeuchteMax OR *)diStatusFrischluftFeuchteMin OR diStatusFrischluftTempMax OR diStatusFrischluftTempMin) AND
		Betriebsparameter.Ausstattung.SensorFrischluft, VerzZeit := Betriebsparameter.Allgemein.VerzoegerungFehler,
		Quit := hmiButtons.QuitFehler, Tick := sekTick, Mode := 1);
		alarmFehler[FEHLER_SENSOR_FRISCHLUFT]	:= fbLascoFehl_15.FehlerOut;

		fbLascoFehl_16(FehlerIn := ((*diStatusDachluftFeuchteMax OR *)diStatusDachluftFeuchteMin OR diStatusDachluftTempMax OR diStatusDachluftTempMin) AND
		Betriebsparameter.Ausstattung.SensorDachluft, VerzZeit := Betriebsparameter.Allgemein.VerzoegerungFehler,
		Quit := hmiButtons.QuitFehler, Tick := sekTick, Mode := 1);
		alarmFehler[FEHLER_SENSOR_DACHLUFT]	:= fbLascoFehl_16.FehlerOut;

		fbLascoFehl_17(FehlerIn := ((*diStatusTrockenluftFeuchteMax OR *)diStatusTrockenluftFeuchteMin OR diStatusTrockenluftTempMax OR diStatusTrockenluftTempMin) AND
		Betriebsparameter.Ausstattung.SensorTrockenluft, VerzZeit := Betriebsparameter.Allgemein.VerzoegerungFehler,
		Quit := hmiButtons.QuitFehler, Tick := sekTick, Mode := 1);
		alarmFehler[FEHLER_SENSOR_TROCKENLUFT]	:= fbLascoFehl_17.FehlerOut;

		fbLascoFehl_18(FehlerIn := ((*diStatusAbluftFeuchteMax OR *)diStatusAbluftFeuchteMin OR diStatusAbluftTempMax OR diStatusAbluftTempMin) AND
		Betriebsparameter.Ausstattung.SensorAbluft,VerzZeit := Betriebsparameter.Allgemein.VerzoegerungFehler,
		Quit := hmiButtons.QuitFehler, Tick := sekTick, Mode := 1);
		alarmFehler[FEHLER_SENSOR_ABLUFT]	:= fbLascoFehl_18.FehlerOut;

		fbLascoFehl_19(FehlerIn := Betriebsparameter.Ausstattung.Entfeuchter AND
		((*diStatusEintrittFeuchteMax OR *)diStatusEintrittFeuchteMin OR diStatusEintrittTempMax OR diStatusEintrittTempMin),
		VerzZeit := Betriebsparameter.Allgemein.VerzoegerungFehler, Quit := hmiButtons.QuitFehler, Tick := sekTick, Mode := 1);
		alarmFehler[FEHLER_SENSOR_EINTRITT]	:= fbLascoFehl_19.FehlerOut;

		alarmFehler[FEHLER_SENSOR_AUSTRITT]	:= FALSE;	//Fehler Sensor Austritt nur als Warnung generieren

		fbLascoFehl_20(FehlerIn := (diStatusLuftgeschwDrahtbruch OR diStatusLuftgeschwMax OR diStatusLuftgeschwMin) AND Betriebsparameter.Ausstattung.SensorLuftgeschwindigkeit,
		VerzZeit := Betriebsparameter.Allgemein.VerzoegerungFehler, Quit := hmiButtons.QuitFehler, Tick := sekTick, Mode := 1);
		alarmFehler[FEHLER_SENSOR_LUFTGESCHW]	:= fbLascoFehl_20.FehlerOut;

		fbLascoFehl_21(FehlerIn := (diStatusDifferenzdruckMax OR diStatusDifferenzdruckMin) AND Betriebsparameter.Ausstattung.SensorKanaldruck,
		VerzZeit := Betriebsparameter.Allgemein.VerzoegerungFehler, Quit := hmiButtons.QuitFehler, Tick := sekTick, Mode := 1);
		alarmFehler[FEHLER_SENSOR_KANALDRUCK]	:= fbLascoFehl_21.FehlerOut;

		fbLascoFehl_22(FehlerIn := Betriebsparameter.Ausstattung.Entfeuchter AND (diStatusNiederdruckMaxMod1 OR diStatusNiederdruckMinMod1),
		VerzZeit := Betriebsparameter.Allgemein.VerzoegerungFehler, Quit := hmiButtons.QuitFehler, Tick := sekTick, Mode := 1);
		alarmFehler[FEHLER_SENSOR_NIEDERDRUCK_MOD1]	:= fbLascoFehl_22.FehlerOut;

		fbLascoFehl_23(FehlerIn := Betriebsparameter.Ausstattung.Entfeuchter AND gModul2Vorhanden AND (diStatusNiederdruckMaxMod2 OR diStatusNiederdruckMinMod2),
		VerzZeit := Betriebsparameter.Allgemein.VerzoegerungFehler, Quit := hmiButtons.QuitFehler, Tick := sekTick, Mode := 1);
		alarmFehler[FEHLER_SENSOR_NIEDERDRUCK_MOD2]	:= fbLascoFehl_23.FehlerOut;

		fbLascoFehl_24(FehlerIn := Betriebsparameter.Ausstattung.Entfeuchter AND (diStatusHochdruckMaxMod1 OR diStatusHochdruckMinMod1),
		VerzZeit := Betriebsparameter.Allgemein.VerzoegerungFehler, Quit := hmiButtons.QuitFehler, Tick := sekTick, Mode := 1);
		alarmFehler[FEHLER_SENSOR_HOCHDRUCK_MOD1]	:= fbLascoFehl_24.FehlerOut;

		fbLascoFehl_25(FehlerIn := Betriebsparameter.Ausstattung.Entfeuchter AND gModul2Vorhanden AND (diStatusHochdruckMaxMod2 OR diStatusHochdruckMinMod2),
		VerzZeit := Betriebsparameter.Allgemein.VerzoegerungFehler, Quit := hmiButtons.QuitFehler, Tick := sekTick, Mode := 1);
		alarmFehler[FEHLER_SENSOR_HOCHDRUCK_MOD2]	:= fbLascoFehl_25.FehlerOut;

		//32) Fehler Endlagen Bypassklappe
		alarmFehler[FEHLER_ENDLAGEN_BYPASSKLAPPE]		:= Aktoren.VentUndKlappen.FehlerLaufzeitBypass AND Betriebsparameter.Ausstattung.Bypassklappe;

		//33) Fehler Endlagen Umschaltklappe 1
		alarmFehler[FEHLER_ENDLAGEN_UMSCHALTKLAPPE1]	:= Aktoren.VentUndKlappen.FehlerLaufzeitUmschaltkl1 AND Betriebsparameter.Ausstattung.Umschaltklappe1;

		//34) Fehler Endlagen Umschaltklappe 2
		alarmFehler[FEHLER_ENDLAGEN_UMSCHALTKLAPPE2]	:= Aktoren.VentUndKlappen.FehlerLaufzeitUmschaltkl2 AND Betriebsparameter.Ausstattung.Umschaltklappe2;

		//35) Fehler Endlagen Boxenklappe 1
		alarmFehler[FEHLER_ENDLAGEN_BOXENKLAPPE_1]		:= Aktoren.VentUndKlappen.FehlerLaufzeitKlappeBox1;

		//36) Fehler Endlagen Boxenklappe 2
		alarmFehler[FEHLER_ENDLAGEN_BOXENKLAPPE_2]		:= Aktoren.VentUndKlappen.FehlerLaufzeitKlappeBox2;

		//37) Fehler Endlagen Boxenklappe 3
		alarmFehler[FEHLER_ENDLAGEN_BOXENKLAPPE_3]		:= Aktoren.VentUndKlappen.FehlerLaufzeitKlappeBox3;

		//38) Fehler Endlagen Boxenklappe 4
		alarmFehler[FEHLER_ENDLAGEN_BOXENKLAPPE_4]		:= Aktoren.VentUndKlappen.FehlerLaufzeitKlappeBox4;

		//39) Fehler Endlagen Boxenklappe 5
		alarmFehler[FEHLER_ENDLAGEN_BOXENKLAPPE_5]		:= Aktoren.VentUndKlappen.FehlerLaufzeitKlappeBox5;

		//40) Fehler Endlagen Boxenklappe 6
		alarmFehler[FEHLER_ENDLAGEN_BOXENKLAPPE_6]		:= Aktoren.VentUndKlappen.FehlerLaufzeitKlappeBox6;

		//41) Fehler Endlagen Abluftklappe
		alarmFehler[FEHLER_ENDLAGEN_ABLUFTKLAPPE]		:= Aktoren.Abluftklappe.FehlerLaufzeit;

		//42) Fehler Temperatur Eintritt zu hoch
		alarmFehler[FEHLER_EINTRITT_TEMP_ZU_HOCH]		:= (gStatusAnlage.EintrittTemperatur > Betriebsparameter.Kompressor1.EintrittTempMax) AND
		Betriebsparameter.Ausstattung.Entfeuchter AND Boxen.FreigabeLuftentfeuchter;

		//43) Fehler Temperatur Eintritt zu niedrig
		alarmFehler[FEHLER_EINTRITT_TEMP_ZU_NIEDRIG]	:= (gStatusAnlage.EintrittTemperatur < Betriebsparameter.Kompressor1.EintrittTempMin) AND
		Betriebsparameter.Ausstattung.Entfeuchter AND Boxen.FreigabeLuftentfeuchter;

		//44) Fehler Laufzeit Pumpdown Kompressor Modul 1
		alarmFehler[FEHLER_LZ_PUMPDOWN_MOD1]			:= Aktoren.KompressorModul1.FehlerPumpdown;

		//45) Fehler Laufzeit Pumpdown Kompressor Modul 2
		alarmFehler[FEHLER_LZ_PUMPDOWN_MOD2]			:= Aktoren.KompressorModul2.FehlerPumpdown AND gModul2Vorhanden;

		//46) Drehfeldüberwachung (Nur bei 3.04 Plus vorhanden)
		IF hmiStatus.NameSteuerung = 3 THEN
			alarmFehler[FEHLER_DREHFELD]	:= NOT diDrehfeldIstKorrekt AND NOT alarmSystem[FEHLER_KOMMUNIKATION_DISPLAY_IO];
		ELSE
			alarmFehler[FEHLER_DREHFELD]	:= FALSE;
		END_IF

		//47) Störmeldung Entfeuchter Fremdgeräte
		fbLascoFehl_29(FehlerIn := Betriebsparameter.Ausstattung.EntfeuchterFremd AND diEntfeuchterFremdStoerung,
		VerzZeit := Betriebsparameter.Allgemein.VerzoegerungFehler, Quit := hmiButtons.QuitFehler, Tick := sekTick, Mode := 2);
		alarmFehler[FEHLER_ENTF_FREMD_STOERMELDUNG]			:= fbLascoFehl_29.FehlerOut;

		//48) Fehler Betriebsmeldung Entfeuchter Fremdgerät
		alarmFehler[FEHLER_ENTF_FREMD_BETRMLDG]			:= Betriebsparameter.Ausstattung.EntfeuchterFremd AND Aktoren.EntfeuchterFremd.FehlerBetriebsmldg; //V2.1.2

		//=======================================================================================================================================================
		//WARNUNGEN ------------------------------ WARNUNGEN ------------------------------ WARNUNGEN ------------------------------ WARNUNGEN ------------------
		//=======================================================================================================================================================

		//00) Warnung wenn Hochdruck Modul 1 zu hoch (Register verschmutzt, Ansaugtemperatur zu hoch oder zu wenig Luftmenge
		fbLascoFehl_26(FehlerIn := gStatusAnlage.Betrieb AND (gStatusAnlage.HochdruckModul1 > Betriebsparameter.Kompressor1.HochdruckMax) AND NOT
		Aktoren.KompressorModul1.KlappenumschaltungAkiv,
		VerzZeit := Betriebsparameter.Allgemein.VerzoegerungWarnungen, Quit := hmiButtons.QuitFehler, Tick := sekTick, Mode := 0);
		alarmWarnung[WARNUNG_HOCHDRUCK_MAX_MOD1]	:= fbLascoFehl_26.FehlerOut;

		//01) Warnung wenn Hochdruck Modul 2 zu hoch (Register verschmutzt, Ansaugtemperatur zu hoch oder zu wenig Luftmenge
		fbLascoFehl_27(FehlerIn := gModul2Vorhanden AND gStatusAnlage.Betrieb AND
		(gStatusAnlage.HochdruckModul2 > Betriebsparameter.Kompressor1.HochdruckMax) AND NOT Aktoren.KompressorModul2.KlappenumschaltungAkiv,
		VerzZeit := Betriebsparameter.Allgemein.VerzoegerungWarnungen, Quit := hmiButtons.QuitFehler, Tick := sekTick, Mode := 0);
		alarmWarnung[WARNUNG_HOCHDRUCK_MAX_MOD2]	:= fbLascoFehl_27.FehlerOut;

		//02) Warnung Sensor Austritt
		fbLascoFehl_28(FehlerIn := diStatusAustrittFeuchteMax OR diStatusAustrittFeuchteMin OR diStatusAustrittTempMax OR diStatusAustrittTempMin,
		VerzZeit := Betriebsparameter.Allgemein.VerzoegerungFehler, Quit := hmiButtons.QuitFehler, Tick := sekTick, Mode := 1);
		alarmWarnung[WARNUNG_SENSOR_AUSTRITT]	:= fbLascoFehl_28.FehlerOut;

		//03) Warnung Heizrregister Frostschutz aktiv
		alarmWarnung[WARNUNG_HEIZREGISTER_FROSTSCHUTZ] := diHeizregisterFrostschutz;

		//==================================================================================================================================================================
		//Fehlerausgang
		//==================================================================================================================================================================

		IF (gStatusAnlage.Betrieb OR gAktModus = STILLSTAND) THEN
			doTrocknungStoerung 	:= gStatusAnlage.Fehler.SummeFehler;
		ELSE
			doTrocknungStoerung	:= FALSE;
		END_IF

	END_IF

	//00 - 04 Systemfehler

	//alarmSystem[FEHLER_KOMMUNIKATION_DISPLAY_IO]	:= ; Wird in den IO-Mappings erzeugt.
	alarmSystem[FEHLER_IO_TEST_NICHT_FERTIG]		:= NOT Nutzungsdaten.Allgemein.IoTestAbgeschlossen;

	//Fehlerquittierung rücksetzen
	TON_Fehlerquittierung.IN	:= hmiButtons.QuitFehler;
	TON_Fehlerquittierung.PT	:= UDINT_TO_TIME(CONST_VERZ_QUIT);
	TON_Fehlerquittierung();

	IF (TON_Fehlerquittierung.Q) THEN
		hmiButtons.QuitFehler	:= FALSE;
	END_IF

	//Gruppenalarme bilden
	//********************

	gStatusAnlage.Fehler.SummeFehler := FALSE;
	gStatusAnlage.Fehler.FehlerNr	 := 0;
	ilen := (SIZEOF(alarmFehler) / SIZEOF(alarmFehler[0])) - 1;
	FOR i := 0 TO ilen DO
		IF (alarmFehler[i] = TRUE) THEN
			gStatusAnlage.Fehler.SummeFehler 	:= TRUE;
			gStatusAnlage.Fehler.FehlerNr		:= i + 1;
			EXIT;
		END_IF
	END_FOR

	gStatusAnlage.Fehler.SummeWarnung := FALSE;
	gStatusAnlage.Fehler.WarnungNr		 := 0;
	ilen := (SIZEOF(alarmWarnung) / SIZEOF(alarmWarnung[0])) - 1;
	FOR i := 0 TO ilen DO
		IF (alarmWarnung[i] = 1) THEN
			gStatusAnlage.Fehler.SummeWarnung 	:= TRUE;
			gStatusAnlage.Fehler.WarnungNr		:= i + 1;
			EXIT;
		END_IF
	END_FOR

	gStatusAnlage.Fehler.SummeSystem := FALSE;
	ilen := (SIZEOF(alarmSystem) / SIZEOF(alarmSystem[0])) - 1;
	FOR i := 0 TO ilen DO
		IF (alarmSystem[i] = 1) THEN
			gStatusAnlage.Fehler.SummeSystem := TRUE;
			EXIT;
		END_IF
	END_FOR

	init	:= TRUE;

END_PROGRAM
```

#### Alarm.var - Lokale Variablen
```iecst
(*============================================================================================================================================*)
(*======================================== FUNKTIONSBAUSTEINE ===============================================================================*)
VAR
	eUhr : fbLascoEUhr;
	fbLascoZdxx_0 : fbLascoZdxx;
	TON_Fehlerquittierung : TON;
	fbLascoFehl_0 : fbLascoFehl;
	fbLascoFehl_1 : fbLascoFehl;
	fbLascoFehl_2 : fbLascoFehl;
	fbLascoFehl_3 : fbLascoFehl;
	fbLascoFehl_4 : fbLascoFehl;
	fbLascoFehl_5 : fbLascoFehl;
	fbLascoFehl_6 : fbLascoFehl;
	fbLascoFehl_7 : fbLascoFehl;
	fbLascoFehl_8 : fbLascoFehl;
	fbLascoFehl_9 : fbLascoFehl;
	fbLascoFehl_10 : fbLascoFehl;
	fbLascoFehl_11 : fbLascoFehl;
	fbLascoFehl_12 : fbLascoFehl;
	fbLascoFehl_13 : fbLascoFehl;
	fbLascoFehl_14 : fbLascoFehl;
	fbLascoFehl_15 : fbLascoFehl;
	fbLascoFehl_16 : fbLascoFehl;
	fbLascoFehl_17 : fbLascoFehl;
	fbLascoFehl_18 : fbLascoFehl;
	fbLascoFehl_19 : fbLascoFehl;
	fbLascoFehl_20 : fbLascoFehl;
	fbLascoFehl_21 : fbLascoFehl;
	fbLascoFehl_22 : fbLascoFehl;
	fbLascoFehl_23 : fbLascoFehl;
	fbLascoFehl_24 : fbLascoFehl;
	fbLascoFehl_25 : fbLascoFehl;
	fbLascoFehl_26 : fbLascoFehl;
	fbLascoFehl_27 : fbLascoFehl;
	fbLascoFehl_28 : fbLascoFehl;
	fbLascoFehl_29 : fbLascoFehl;
END_VAR
(*============================================================================================================================================*)
(*======================================== LOKALE VARIABLEN ==================================================================================*)
VAR
	init : BOOL;
	sekTick : BOOL;
	ilen : USINT;
	i : USINT;
END_VAR
(*============================================================================================================================================*)
(*======================================== KONSTANTEN ==================================================================================*)
VAR
	CONST_VERZ_STOERUNG_ENTF_FREMD : {REDUND_UNREPLICABLE} UDINT := 60; (*Verzögerungszeit Störungseingang Entfeuchter Fremd [sek]*)
	CONST_VERZ_QUIT : {REDUND_UNREPLICABLE} UDINT := 2000; (*Verzögerung, bevor die Fehlerquittierung wieder rückgesetzt wird*)
END_VAR
```

### Alarmsys.var - Fehler und Warnungen
```iecst
VAR
	alarmWarnung : ARRAY[0..29] OF BOOL := [30(FALSE)];
	alarmFehler : ARRAY[0..49] OF BOOL := [50(FALSE)];
	alarmSystem : ARRAY[0..4] OF BOOL := [5(FALSE)];
END_VAR
```

### Package Logical/Ablaufsteuerung - Ablaufsteuerung, Schrittkette

### Program Logical/Ablaufsteuerung/Ablaufstrg (IEC) - Ablaufsteuerung Hauptprogramm

#### Ablaufstrg.st - Zyklischer Code
```iecst
PROGRAM _INIT

	stateEntry			:= TRUE;
	nextModus			:= STILLSTAND;

END_PROGRAM

PROGRAM _CYCLIC

	//Zeitticks generieren
	zdxxSekunden(IN		:= Echtzeit.Sekunde);
	sekTick				:= zdxxSekunden.Q;
	zdxxMinuten(IN 		:= Echtzeit.Minute);
	minTick				:= zdxxMinuten.Q;
	zdxxStunden(IN		:= Echtzeit.Stunde);
	stdTick				:= zdxxStunden.Q;
	zdxxTage(IN			:= Echtzeit.Tag);
	TagTick				:= zdxxTage.Q;

	//Schrittschaltwerk Ablaufsteuerung
	//=================================

	gAktModus := nextModus;

	actionUpdateStatus;

	CASE gAktModus OF

		//********************************************************************************************************************************************************************************************************
		STILLSTAND:

			//*** State entry ***
			IF (stateEntry) THEN
				stateEntry 					:= FALSE;
				Strombegrenzung.Freigabe	:= FALSE;
				Tarifabschaltung.Freigabe	:= FALSE;
			END_IF

			//*** State during	***
			actionStillstand;

			//*** State exit ***

			//Startsignal
			IF (gCmdAnlage.Start AND gCmdAnlage.Auto) THEN
				nextModus 	:= BETRIEB;
				stateEntry 	:= TRUE;
			//Stromausfall im Betrieb
			ELSIF (Nutzungsdaten.Allgemein.LetzterModus = BETRIEB)  THEN
				nextModus 	:= BETRIEB;
				stateEntry 	:= TRUE;
			//Testbetrieb
			ELSIF (gCmdAnlage.Test AND NOT gCmdAnlage.Auto) THEN
				nextModus 	:= IOTEST;
				stateEntry 	:= TRUE;
			ELSE
				nextModus 	:= gAktModus;
			END_IF

		//********************************************************************************************************************************************************************************************************
		BETRIEB:

			//*** State entry ***
			IF (stateEntry) THEN
				stateEntry 								:= FALSE;
				hmiNutzungsdaten.Allgemein.LetzterModus	:= BETRIEB;
			END_IF

			//*** State during	***
			actionBetrieb;

			//Funktionsbaustein Strombegrenzung
			Strombegrenzung.Freigabe	:= TRUE;
			Strombegrenzung.AktZeit		:= Echtzeit.StdMin;

			//Funktionsbaustein Tarifabschaltung
			Tarifabschaltung.Freigabe	:= TRUE;
			Tarifabschaltung.AktZeit	:= Echtzeit.StdMin;

			//*** State exit ***

			//Stopp
			IF (gCmdAnlage.Stop) THEN
				hmiNutzungsdaten.Allgemein.LetzterModus	:= STILLSTAND;
				nextModus		:= STILLSTAND;
				stateEntry		:= TRUE;
			ELSE
				nextModus		:= gAktModus;
			END_IF

			//********************************************************************************************************************************************************************************************************
		IOTEST:

			//*** State entry ***
			IF (stateEntry) THEN
				stateEntry 		:= FALSE;
			END_IF

			//*** State during	***
			gStatusAnlage.Aktor[AKTOR_SCHRITTKETTE] := STATUS_TESTBETRIEB;

			//*** State exit ***

			//Testbetrieb abgeschlossen
			IF (NOT gCmdAnlage.Test) THEN
				nextModus 	:= STILLSTAND;
				stateEntry 	:= TRUE;
			ELSE
				nextModus 	:= gAktModus;
			END_IF

	END_CASE

	//Funktionsbausteine aufrufen
	//***************************
	Boxen();
	Aktoren.Abluftklappe();
	Aktoren.Abluftventilator();
	Aktoren.Brandschutzklappe();
	Aktoren.Heizregister();
	Aktoren.EntfeuchterFremd();
	Aktoren.KompressorModul1();
	Aktoren.KompressorModul2();
	Aktoren.Notstromaggregat();
	Aktoren.OelsumpfheizungModul1();
	Aktoren.OelsumpfheizungModul2();
	Aktoren.Scheitholzofen();
	Aktoren.VentUndKlappen();
	Aktoren.Warmluftofen();

	fbSchlechtwetterBox1();
	fbSchlechtwetterBox2();
	fbSchlechtwetterBox3();
	fbSchlechtwetterBox4();
	fbSchlechtwetterBox5();
	fbSchlechtwetterBox6();

	//Umschaltung Dachluft/Umluft je nach Ausstattung
	fbEntfUmschaltung_0.Freigabe					:= Betriebsparameter.Ausstattung.Umschaltklappe1 OR Betriebsparameter.Ausstattung.Umschaltklappe2;
	fbEntfUmschaltung_0.AbluftTemp					:= gStatusAnlage.AbluftTemperatur;
	fbEntfUmschaltung_0.DachluftTemp				:= gStatusAnlage.DachluftTemperatur;
	fbEntfUmschaltung_0.FrischluftTemp				:= gStatusAnlage.FrischluftTemperatur;
	fbEntfUmschaltung_0.FrischlDachlTempUmschaltung	:= Betriebsparameter.Umschaltklappen.TemperaturUmschaltung;
	fbEntfUmschaltung_0.DifferenzTempUmschaltung	:= Betriebsparameter.Umschaltklappen.TempDifferenzUmschaltung;
	fbEntfUmschaltung_0.Hysterese					:= Betriebsparameter.Umschaltklappen.Hysterese;
	fbEntfUmschaltung_0.SensorAbluftVhd				:= Betriebsparameter.Ausstattung.SensorAbluft;
	fbEntfUmschaltung_0.SensorDachluftVhd			:= Betriebsparameter.Ausstattung.SensorDachluft;
	fbEntfUmschaltung_0.SensorFrischluftVhd			:= Betriebsparameter.Ausstattung.SensorFrischluft;
	fbEntfUmschaltung_0.StatusSensorAbluftOk		:= NOT alarmFehler[FEHLER_SENSOR_ABLUFT];
	fbEntfUmschaltung_0.StatusSensorDachluftOk		:= NOT alarmFehler[FEHLER_SENSOR_DACHLUFT];
	fbEntfUmschaltung_0.StatusSensorFrischluftOk	:= NOT alarmFehler[FEHLER_SENSOR_FRISCHLUFT];
	fbEntfUmschaltung_0.Umschaltverz				:= Betriebsparameter.Umschaltklappen.Umschaltverzoegerung;
	fbEntfUmschaltung_0();

	//Tarifabschaltung
	Tarifabschaltung.StartMin1	:= Betriebsparameter.Tarifabschaltung.Zeitfenster.StartMin;
	Tarifabschaltung.StartStd1	:= Betriebsparameter.Tarifabschaltung.Zeitfenster.StartStd;
	Tarifabschaltung.StoppMin1	:= Betriebsparameter.Tarifabschaltung.Zeitfenster.StoppMin;
	Tarifabschaltung.StoppStd1	:= Betriebsparameter.Tarifabschaltung.Zeitfenster.StoppStd;
	Tarifabschaltung.VorlaufzeitLuftaufbMin	:= Betriebsparameter.Tarifabschaltung.VorlaufzeitAbschaltungLuftaufb;
	Tarifabschaltung();

	//Strombegrenzung
	//Start- und Stoppzeiten in Format "hhmm" umrechnen
	loc_StrombegrStart1			:= (Betriebsparameter.Strombegrenzung.Zeitfenster.StartStd * 100) + Betriebsparameter.Strombegrenzung.Zeitfenster.StartMin;
	loc_StrombegrStopp1			:= (Betriebsparameter.Strombegrenzung.Zeitfenster.StoppStd * 100) + Betriebsparameter.Strombegrenzung.Zeitfenster.StoppMin;
	Strombegrenzung.StartZeit1	:= loc_StrombegrStart1;
	Strombegrenzung.StoppZeit1	:= loc_StrombegrStopp1;
	Strombegrenzung();

END_PROGRAM
```

#### Ablaufstrg.var - Lokale Variablen
```iecst
(*==================================================================================================================================================================*)
(*===================================================   FUNKTIONSBAUSTEINE =========================================================================================*)
VAR
	zdxxSekunden : {REDUND_UNREPLICABLE} fbLascoZdxx;
	zdxxMinuten : {REDUND_UNREPLICABLE} fbLascoZdxx;
	zdxxTage : {REDUND_UNREPLICABLE} fbLascoZdxx;
	zdxxStunden : {REDUND_UNREPLICABLE} fbLascoZdxx;
END_VAR
(*==================================================================================================================================================================*)
(*===================================================   ZEITTICKS  ====================================================================================================*)
VAR
	sekTick : {REDUND_UNREPLICABLE} BOOL;
	minTick : {REDUND_UNREPLICABLE} BOOL;
	stdTick : {REDUND_UNREPLICABLE} BOOL;
	TagTick : {REDUND_UNREPLICABLE} BOOL;
END_VAR
(*==================================================================================================================================================================*)
(*===================================================   SONSTIGE  ====================================================================================================*)
VAR
	nextModus : {REDUND_UNREPLICABLE} enumBetriebsmodus;
	stateEntry : {REDUND_UNREPLICABLE} BOOL;
	fbEntfUmschaltung_0 : {REDUND_UNREPLICABLE} fbBoxenUmschaltung;
	loc_StrombegrStart1 : {REDUND_UNREPLICABLE} UINT;
	loc_StrombegrStopp1 : {REDUND_UNREPLICABLE} UINT;
END_VAR
```
